(* PLC project SPS_Demonstrator, Beckhoff Automation GmbH TwinCAT PLC Control 3.5.21.30 *)
(* stored: creationDateTime 2026-04-30T11:55:43.4526457, modificationDateTime 2026-04-30T11:55:43.4526457 *)

PROGRAM HRL_SkillSet
VAR
//Hochregallager Skillset	
	//HRL CombinedSkill_Auslagerung
	{attribute 'OPC.UA.DA':= '1'}
	HRL_NMethod_Auslagern : HRL_NMethod_Auslagern;
	bAuslagernAktiv : BOOL := FALSE;
	//HRL Conveyorbelt Skills
	{attribute 'OPC.UA.DA':= '1'}
	HRL_Skill_CB_MoveForwards: HRL_CB_AS_HorizontalMoveSensors; //Movement to Store-Out some goods on the Conveyorbelt
	{attribute 'OPC.UA.DA':= '1'}
	HRL_Skill_CB_MoveBackwards : HRL_CB_AS_HorizontalMoveSensors; //Movement to Store-In some goods on the Conveyorbelt
	
	//HRL RGB Skills
	{attribute 'OPC.UA.DA':= '1'}
	HRL_Skill_RGB_MoveBackwards : HRL_RGB_AS_HorizontalMoveSensors;	
	{attribute 'OPC.UA.DA':= '1'}
	HRL_Skill_RGB_MoveForwards : HRL_RGB_AS_HorizontalMoveSensors;	
	{attribute 'OPC.UA.DA':= '1'}
	HRL_Skill_RGB_MoveVerticalForwards : HRL_RGB_AS_VerticalMoveEncoders;	
	{attribute 'OPC.UA.DA':= '1'}
	HRL_Skill_RGB_MoveVerticalBackwards : HRL_RGB_AS_VerticalMoveEncoders;
	{attribute 'OPC.UA.DA':= '1'}
	HRL_Skill_RGB_MoveHorizontalForwards : HRL_RGB_AS_HorizontalMoveEncoders;	
	{attribute 'OPC.UA.DA':= '1'}
	HRL_Skill_RGB_MoveHorizontalBackwards : HRL_RGB_AS_HorizontalMoveEncoders;
	
	//Organisation FBs
	HRL_ControlOfOutputs : HRL_ControlOfOutputs;
	HRL_OperatingModes : HRL_OperatingModes;
	HRL_DiagnosisHandler : HRL_DiagnosisHandler;
	bAuslagernTrackingLatched : BOOL := FALSE;
	
	//InitialStateDrives
	HRL_RGB_InitialStateDrive : HRL_RGB_InitialStateDrive;
	
	
//Variablen zur Outputsteuerung
	HRL_CB_forwards : BOOL; //GVL_HRL.HRL_MOT_Foerderband_vorwaerts
	HRL_CB_backwards : BOOL; //GVL_HRL.HRL_MOT_Foerderband_rueckwaerts
	HRL_RGB_Forwards01 : BOOL; //GVL_HRL.HRL_MOT_Ausleger_vorwaerts
	HRL_RGB_Forwards02 : BOOL; //GVL_HRL.HRL_MOT_Ausleger_vorwaerts
	HRL_RGB_Backwards01 : BOOL; //GVL_HRL.HRL_MOT_Ausleger_rueckwaerts
	HRL_RGB_Backwards02 : BOOL; //GVL_HRL.HRL_MOT_Ausleger_rueckwaerts	
	HRL_RGB_VertikalDown01 : BOOL; //GVL_HRL.HRL_MOT_vertikal_runter		
	HRL_RGB_VertikalDown02 : BOOL; //GVL_HRL.HRL_MOT_vertikal_runter
	HRL_RGB_VertikalUp01 : BOOL; //GVL_HRL.HRL_MOT_vertikal_hoch
	HRL_RGB_VertikalUp02 : BOOL; //GVL_HRL.HRL_MOT_vertikal_hoch
	HRL_RGB_HorizontalForwards01 : BOOL; //GVL_HRL.HRL_MOT_horizontal_zum_Regal	
	HRL_RGB_HorizontalForwards02 : BOOL; //GVL_HRL.HRL_MOT_horizontal_zum_Regal	
	HRL_RGB_HorizontalBackwards01 : BOOL; //GVL_HRL.HRL_MOT_horizontal_zum_Foerderband
	HRL_RGB_HorizontalBackwards02 : BOOL; //GVL_HRL.HRL_MOT_horizontal_zum_Foerderband
//OutputVariablen für Init-Fahrt	
	Init_SRM_MotorBackwards : BOOL;
	Init_SRM_MotorForwards : BOOL;
	Init_RGB_VerticalUp : BOOL;
	Init_RGB_VerticalDown : BOOL;
	Init_RGB_HorizontalForwards : BOOL;
	Init_RGB_HorizontalBackwards : BOOL;
	
//Time Constraints
	TIME_TSR : TIME := T#150MS;
//Encoder Values for InitialStateDrive
	HRL_RGB_ET_Vertical01 : UDINT;
	HRL_RGB_ET_Vertical02 : UDINT;
	HRL_RGB_ET_Horizontall01 : UDINT;
	HRL_RGB_ET_Horizontall02 : UDINT;
	
	//GEMMA_Mappings
	sCurrentGemmaState : STRING(80) := '';
    sLastNonFailureGemmaState : STRING(80) := '';
    rtD2 : R_TRIG;
END_VAR

VAR_INPUT
	//Variablensetzung: Sollte später über SkillOA eingesetzt werden ODER Hard in SPS codiert (Diskussionspunkt)
	ResetButton: BOOL;
	StartButton: BOOL;
	ConfirmationButton: BOOL;
END_VAR

                  (* === Simulations-Override *)
IF GVL_Sim.bSimMode THEN
    GVL.diNotAus_Kanal_A                  := GVL_Sim.diNotAus_Kanal_A;
    GVL.diNotAus_Kanal_B                  := GVL_Sim.diNotAus_Kanal_B;
    GVL_HRL.HRL_Enc_horizontal_I1          := GVL_HRL_Sim.HRL_Enc_horizontal_I1;
    GVL_HRL.HRL_Enc_horizontal_I2          := GVL_HRL_Sim.HRL_Enc_horizontal_I2;
    GVL_HRL.HRL_Enc_vertikal_I1            := GVL_HRL_Sim.HRL_Enc_vertikal_I1;
    GVL_HRL.HRL_Enc_vertikal_I2            := GVL_HRL_Sim.HRL_Enc_vertikal_I2;
    // GVL_HRL - Digitaleingänge (BOOL)
    GVL_HRL.HRL_Ref_Taster_horizontal      := GVL_HRL_Sim.HRL_Ref_Taster_horizontal;
    GVL_HRL.HRL_LS_innen                   := GVL_HRL_Sim.HRL_LS_innen;
    GVL_HRL.HRL_LS_aussen                  := GVL_HRL_Sim.HRL_LS_aussen;
    GVL_HRL.HRL_Ref_Taster_vertikal        := GVL_HRL_Sim.HRL_Ref_Taster_vertikal;
    GVL_HRL.HRL_Spursensor_1_unten         := GVL_HRL_Sim.HRL_Spursensor_1_unten;
    GVL_HRL.HRL_Spursensor_2_oben          := GVL_HRL_Sim.HRL_Spursensor_2_oben;
    GVL_HRL.HRL_Ref_Taster_Ausleger_vorne  := GVL_HRL_Sim.HRL_Ref_Taster_Ausleger_vorne;
    GVL_HRL.HRL_Ref_Taster_Ausleger_hinten := GVL_HRL_Sim.HRL_Ref_Taster_Ausleger_hinten;
END_IF
(* ============================================================================= *)
HRL_OperatingModes(
    Start := StartButton,
    Stop := NOT (((GVL.diNotAus_Kanal_A) AND (GVL.diNotAus_Kanal_B))),
    Reset := ResetButton,
    Schalter := ConfirmationButton,
    Schrittkette_GS := ((HRL_RGB_InitialStateDrive.ResetMethodCall_SRM) AND (HRL_RGB_InitialStateDrive.ResetMethodCall_RGB_Horizontal) AND (HRL_RGB_InitialStateDrive.ResetMethodCall_RGB_Vertical)),
    Count1 := HRL_RGB_InitialStateDrive.Count_SRM_MotorBackw,
    Count2 := HRL_RGB_InitialStateDrive.Count_SRM_MotorForw,
    Alt_abort := OPCUA.Alt_abort,
    Err_detected := HRL_DiagnosisHandler.Err_detected,
    Diag_finished := HRL_DiagnosisHandler.Diag_finished,
    Alt_found := HRL_DiagnosisHandler.Alt_found,
    Cycle_finished := OPCUA.Cycle_finished
);


HRL_NMethod_Auslagern(
    ESS_OK := ((GVL.diNotAus_Kanal_A) AND (GVL.diNotAus_Kanal_B)),
    AutomaticMode := HRL_OperatingModes.F1,

    HRL_Enc_horizontal_I1 := GVL_HRL.HRL_Enc_horizontal_I1,
    HRL_Enc_horizontal_I2 := GVL_HRL.HRL_Enc_horizontal_I2,
    HRL_Enc_vertikal_I1 := GVL_HRL.HRL_Enc_vertikal_I1,
    HRL_Enc_vertikal_I2 := GVL_HRL.HRL_Enc_vertikal_I2,

    HRL_Ref_Taster_horizontal := GVL_HRL.HRL_Ref_Taster_horizontal,
    HRL_Ref_Taster_vertikal := GVL_HRL.HRL_Ref_Taster_vertikal,
    HRL_Ref_Taster_Ausleger_vorne := GVL_HRL.HRL_Ref_Taster_Ausleger_vorne,
    HRL_Ref_Taster_Ausleger_hinten := GVL_HRL.HRL_Ref_Taster_Ausleger_hinten,

    HRL_LS_innen := GVL_HRL.HRL_LS_innen,
    HRL_LS_aussen := GVL_HRL.HRL_LS_aussen
);

HRL_DiagnosisHandler(
    Diagnose_gefordert := HRL_OperatingModes.D2,
    ErrorDetectedRaw := HRL_NMethod_Auslagern.Error,
    Reset := ResetButton
);

HRL_RGB_InitialStateDrive(
    MethodCall_InitDrive := HRL_OperatingModes.MethodCall_InitStateDrive,
    ESS := ((GVL.diNotAus_Kanal_A) AND (GVL.diNotAus_Kanal_B)),
    InputInitDriveMode := HRL_OperatingModes.InputVar_InitStateDrive,
    TouchSensor01_SRM := GVL_HRL.HRL_Ref_Taster_Ausleger_hinten,
    TouchSensor02_RGB_vertical := GVL_HRL.HRL_Ref_Taster_vertikal,
    TouchSensor03_RGB_horizontal := GVL_HRL.HRL_Ref_Taster_horizontal,
    TOF_Time_TSR := TIME_TSR,
    InitDriveMode := HRL_OperatingModes.A6
);
Init_SRM_MotorBackwards := HRL_RGB_InitialStateDrive.SRM_MotorBackwards;
HRL_Skill_CB_MoveForwards(
    ESS := ((GVL.diNotAus_Kanal_A) AND (GVL.diNotAus_Kanal_B)),
    LightBarrierSensor_01 := GVL_HRL.HRL_LS_innen,
    LightBarrierSensor_02 := GVL_HRL.HRL_LS_aussen,
    AutomaticMode := HRL_OperatingModes.F1
);
HRL_CB_forwards := HRL_Skill_CB_MoveForwards.DO_MovingConveyorBelt;
HRL_Skill_CB_MoveBackwards(
    ESS := ((GVL.diNotAus_Kanal_A) AND (GVL.diNotAus_Kanal_B)),
    LightBarrierSensor_01 := GVL_HRL.HRL_LS_aussen,
    LightBarrierSensor_02 := GVL_HRL.HRL_LS_innen,
    AutomaticMode := HRL_OperatingModes.F1
);
HRL_CB_backwards := HRL_Skill_CB_MoveBackwards.DO_MovingConveyorBelt;
HRL_Skill_RGB_MoveForwards(
    ESS := ((GVL.diNotAus_Kanal_A) AND (GVL.diNotAus_Kanal_B)),
    TouchSensor01 := GVL_HRL.HRL_Ref_Taster_Ausleger_hinten,
    TouchSensor02 := GVL_HRL.HRL_Ref_Taster_Ausleger_vorne,
    TOF_Time_TSR := TIME_TSR,
    AutomaticMode := HRL_OperatingModes.F1
);
HRL_RGB_Forwards01 := HRL_Skill_RGB_MoveForwards.DO_MovingHorizontalRGB_01;
HRL_Skill_RGB_MoveBackwards(
    ESS := ((GVL.diNotAus_Kanal_A) AND (GVL.diNotAus_Kanal_B)),
    TouchSensor01 := GVL_HRL.HRL_Ref_Taster_Ausleger_vorne,
    TouchSensor02 := GVL_HRL.HRL_Ref_Taster_Ausleger_hinten,
    TOF_Time_TSR := TIME_TSR,
    AutomaticMode := HRL_OperatingModes.F1
);
HRL_RGB_Backwards01 := HRL_Skill_RGB_MoveBackwards.DO_MovingHorizontalRGB_01;
HRL_Skill_RGB_MoveVerticalForwards(
    ESS := ((GVL.diNotAus_Kanal_A) AND (GVL.diNotAus_Kanal_B)),
    TouchSensor01 := GVL_HRL.HRL_Ref_Taster_vertikal,
    EncoderStartPosition01 := GVL_HRL.HRL_Enc_vertikal_I1,
    EncoderStartPosition02 := GVL_HRL.HRL_Enc_vertikal_I2,
    TOF_TSR_TIME := TIME_TSR,
    AutomaticMode := HRL_OperatingModes.F1
);
HRL_RGB_VertikalDown01 := HRL_Skill_RGB_MoveVerticalForwards.DO_MovingVerticalRGB_01;
HRL_Skill_RGB_MoveVerticalBackwards(
    ESS := ((GVL.diNotAus_Kanal_A) AND (GVL.diNotAus_Kanal_B)),
    TouchSensor01 := GVL_HRL.HRL_Ref_Taster_vertikal,
    EncoderStartPosition01 := GVL_HRL.HRL_Enc_vertikal_I1,
    EncoderStartPosition02 := GVL_HRL.HRL_Enc_vertikal_I2,
    TOF_TSR_TIME := TIME_TSR,
    AutomaticMode := HRL_OperatingModes.F1
);
HRL_RGB_VertikalUp02 := HRL_Skill_RGB_MoveVerticalBackwards.DO_MovingVerticalRGB_01;
HRL_Skill_RGB_MoveHorizontalForwards(
    ESS := ((GVL.diNotAus_Kanal_A) AND (GVL.diNotAus_Kanal_B)),
    TouchSensor01 := GVL_HRL.HRL_Ref_Taster_horizontal,
    EncoderStartPosition01 := GVL_HRL.HRL_Enc_horizontal_I1,
    EncoderStartPosition02 := GVL_HRL.HRL_Enc_horizontal_I2,
    TOF_Time_TSR := TIME_TSR,
    AutomaticMode := HRL_OperatingModes.F1
);
HRL_RGB_HorizontalForwards01 := HRL_Skill_RGB_MoveHorizontalForwards.DO_MovingHorizontalRGB_01;
HRL_Skill_RGB_MoveHorizontalBackwards(
    ESS := ((GVL.diNotAus_Kanal_A) AND (GVL.diNotAus_Kanal_B)),
    TouchSensor01 := GVL_HRL.HRL_Ref_Taster_horizontal,
    EncoderStartPosition01 := GVL_HRL.HRL_Enc_horizontal_I1,
    EncoderStartPosition02 := GVL_HRL.HRL_Enc_horizontal_I2,
    TOF_Time_TSR := TIME_TSR,
    AutomaticMode := HRL_OperatingModes.F1
);
HRL_RGB_HorizontalBackwards02 := HRL_Skill_RGB_MoveHorizontalBackwards.DO_MovingHorizontalRGB_01;

bAuslagernAktiv := HRL_NMethod_Auslagern.Busy OR (HRL_NMethod_Auslagern.CurrentStep <> 0);;

HRL_ControlOfOutputs(
    F4 := HRL_OperatingModes.F4,
    F1 := HRL_OperatingModes.F1,
    A2 := HRL_OperatingModes.A2,
    A1 := HRL_OperatingModes.A1,
    A6 := HRL_OperatingModes.A6,
    Start := HRL_OperatingModes.Start,

    CB_forwards :=
        (HRL_CB_forwards AND NOT bAuslagernAktiv)
        OR HRL_NMethod_Auslagern.REQ_CB_forwards,

    CB_backwards :=
        (HRL_CB_backwards AND NOT bAuslagernAktiv)
        OR HRL_NMethod_Auslagern.REQ_CB_backwards,

    RGB_Forwards01 :=
        (HRL_RGB_Forwards01 AND NOT bAuslagernAktiv)
        OR HRL_NMethod_Auslagern.REQ_RGB_Forwards,

    RGB_Forwards02 :=
        HRL_RGB_Forwards02 AND NOT bAuslagernAktiv,

    RGB_Backwards01 :=
        (HRL_RGB_Backwards01 AND NOT bAuslagernAktiv)
        OR HRL_NMethod_Auslagern.REQ_RGB_Backwards,

    RGB_Backwards02 :=
        HRL_RGB_Backwards02 AND NOT bAuslagernAktiv,

    RGB_VertikalDown01 :=
        (HRL_RGB_VertikalDown01 AND NOT bAuslagernAktiv)
        OR HRL_NMethod_Auslagern.REQ_RGB_VerticalDown,

    RGB_VertikalDown02 :=
        HRL_RGB_VertikalDown02 AND NOT bAuslagernAktiv,

    RGB_VertikalUp01 :=
        (HRL_RGB_VertikalUp01 AND NOT bAuslagernAktiv)
        OR HRL_NMethod_Auslagern.REQ_RGB_VerticalUp,

    RGB_VertikalUp02 :=
        HRL_RGB_VertikalUp02 AND NOT bAuslagernAktiv,

    RGB_HorizontalForwards01 :=
        (HRL_RGB_HorizontalForwards01 AND NOT bAuslagernAktiv)
        OR HRL_NMethod_Auslagern.REQ_RGB_HorizontalForward,

    RGB_HorizontalForwards02 :=
        HRL_RGB_HorizontalForwards02 AND NOT bAuslagernAktiv,

    RGB_HorizontalBackwards01 :=
        (HRL_RGB_HorizontalBackwards01 AND NOT bAuslagernAktiv)
        OR HRL_NMethod_Auslagern.REQ_RGB_HorizontalBackward,

    RGB_HorizontalBackwards02 :=
        HRL_RGB_HorizontalBackwards02 AND NOT bAuslagernAktiv,

    Init_RGB_Forwards := Init_SRM_MotorForwards,
    Init_RGB_Backwards := Init_SRM_MotorBackwards,
    Init_RGB_VertikalUp := Init_RGB_VerticalUp,
    Init_RGB_VertikalDown := Init_RGB_VerticalDown,
    Init_RGB_HorizontalForwads := Init_RGB_HorizontalForwards,
    Init_RGB_HorizontalBackwards := Init_RGB_HorizontalBackwards
);
IF GVL_Sim.bSimMode THEN

    // Outputs in Simulationsabbild schreiben
    GVL_HRL_Sim.HRL_MOT_Foerderband_vorwaerts :=
        HRL_ControlOfOutputs.ConveyorBeltForward;

    GVL_HRL_Sim.HRL_MOT_Foerderband_rueckwaerts :=
        HRL_ControlOfOutputs.ConveyorBeltBackward;

    GVL_HRL_Sim.HRL_MOT_Ausleger_vorwaerts :=
        HRL_ControlOfOutputs.RGB_Forwards;

    GVL_HRL_Sim.HRL_MOT_Ausleger_rueckwaerts :=
        HRL_ControlOfOutputs.RGB_Backwards;

    GVL_HRL_Sim.HRL_MOT_vertikal_runter :=
        HRL_ControlOfOutputs.RGB_VerticalDown;

    GVL_HRL_Sim.HRL_MOT_vertikal_hoch :=
        HRL_ControlOfOutputs.RGB_VerticalUp;

    GVL_HRL_Sim.HRL_MOT_horizontal_zum_Regal :=
        HRL_ControlOfOutputs.RGB_HorizontalForward;

    GVL_HRL_Sim.HRL_MOT_horizontal_zum_Foerderband :=
        HRL_ControlOfOutputs.RGB_HorizontalBackward;

    GVL_HRL_Sim.HRL_K1_1_Zaehler_Zuruecksetzen :=
        GVL_HRL.HRL_K1_1_Zaehler_Zuruecksetzen;

    GVL_HRL_Sim.HRL_K1_2_Zaehler_Zuruecksetzen :=
        GVL_HRL.HRL_K1_2_Zaehler_Zuruecksetzen;

ELSE

    // Outputs auf reale Hardware schreiben
    GVL_HRL.HRL_MOT_Foerderband_vorwaerts :=
        HRL_ControlOfOutputs.ConveyorBeltForward;

    GVL_HRL.HRL_MOT_Foerderband_rueckwaerts :=
        HRL_ControlOfOutputs.ConveyorBeltBackward;

    GVL_HRL.HRL_MOT_Ausleger_vorwaerts :=
        HRL_ControlOfOutputs.RGB_Forwards;

    GVL_HRL.HRL_MOT_Ausleger_rueckwaerts :=
        HRL_ControlOfOutputs.RGB_Backwards;

    GVL_HRL.HRL_MOT_vertikal_runter :=
        HRL_ControlOfOutputs.RGB_VerticalDown;

    GVL_HRL.HRL_MOT_vertikal_hoch :=
        HRL_ControlOfOutputs.RGB_VerticalUp;

    GVL_HRL.HRL_MOT_horizontal_zum_Regal :=
        HRL_ControlOfOutputs.RGB_HorizontalForward;

    GVL_HRL.HRL_MOT_horizontal_zum_Foerderband :=
        HRL_ControlOfOutputs.RGB_HorizontalBackward;

END_IF;

//GEMMA-Mappings
IF HRL_OperatingModes.A1 THEN
    sCurrentGemmaState := 'HRL_OperatingModes.A1';
ELSIF HRL_OperatingModes.A2 THEN
    sCurrentGemmaState := 'HRL_OperatingModes.A2';
ELSIF HRL_OperatingModes.A5 THEN
    sCurrentGemmaState := 'HRL_OperatingModes.A5';
ELSIF HRL_OperatingModes.A6 THEN
    sCurrentGemmaState := 'HRL_OperatingModes.A6';
ELSIF HRL_OperatingModes.F1 THEN
    sCurrentGemmaState := 'HRL_OperatingModes.F1';
ELSIF HRL_OperatingModes.F4 THEN
    sCurrentGemmaState := 'HRL_OperatingModes.F4';
ELSIF HRL_OperatingModes.D1 THEN
    sCurrentGemmaState := 'HRL_OperatingModes.D1';
ELSIF HRL_OperatingModes.D3 THEN
    sCurrentGemmaState := 'HRL_OperatingModes.D3';
END_IF;

IF NOT HRL_OperatingModes.D2 THEN
    sLastNonFailureGemmaState := sCurrentGemmaState;
END_IF;

rtD2(CLK := HRL_OperatingModes.D2);

IF rtD2.Q THEN
    OPCUA.LastGEMMAStateBeforeFailure := sLastNonFailureGemmaState;
END_IF;
                
END_PROGRAM

PROGRAM MBS_SkillSet
VAR
//Multibearbeitungsstation Skills
	//MBS Maschine1 (Ofen) Skills	
	{attribute 'OPC.UA.DA':= '1'}
	MBS_Skill_MR01_TransportIn: MBS_MR01_AS_HorizontalMoveSensors;
	{attribute 'OPC.UA.DA':= '1'}
	MBS_Skill_MR01_SecuringWorkpiece: MBS_MR01_AS_SecuringProcess;
	{attribute 'OPC.UA.DA':= '1'}
	MBS_Skill_MR01_HardeningProcess: MBS_MR01_AS_HardeningProcess;
	{attribute 'OPC.UA.DA':= '1'}
	MBS_SkillMR01_ReleaseWorkpiece: MBS_MR01_AS_SecuringProcess;
	{attribute 'OPC.UA.DA':= '1'}
	MBS_Skill_MR01_TransportOut: MBS_MR01_AS_HorizontalMoveSensors;
	
	//MBS Vakuumsauggreifer Skills
	{attribute 'OPC.UA.DA':= '1'}
	MBS_Skill_VGS_PickUpWorkpieceToDmPD: MBS_VSG_AS_SuctionProcess;
	{attribute 'OPC.UA.DA':= '1'}
	MBS_Skill_VGS_PickUpWorkpieceToOven: MBS_VSG_AS_SuctionProcess;
	{attribute 'OPC.UA.DA':= '1'}
	MBS_Skill_VSG_VerticalMove: MBS_VSG_AS_VerticalMove;	
	{attribute 'OPC.UA.DA':= '1'}
	MBS_Skill_VSG_TransportToDmPD: MBS_VSG_AS_HorizontalMove;
	{attribute 'OPC.UA.DA':= '1'}
	MBS_Skill_VSG_TransportToMR01: MBS_VSG_AS_HorizontalMove;
	
	
	//MBS Drehteller mit PushingDevice Skills
	{attribute 'OPC.UA.DA':= '1'}
	MBS_Skill_DmPD_RotateFromVSGtoMR02: MBS_DmPD_AS_RotationMove;
	{attribute 'OPC.UA.DA':= '1'}
	MBS_Skill_DmPD_RotateFromVSGtoCB: MBS_DmPD_AS_RotationMove;
	{attribute 'OPC.UA.DA':= '1'}
	MBS_Skill_DmPD_RotateFromMR02toCB: MBS_DmPD_AS_RotationMove;
	{attribute 'OPC.UA.DA':= '1'}
	MBS_Skill_DmPD_RotateFromMR02toVSG: MBS_DmPD_AS_RotationMove;
	{attribute 'OPC.UA.DA':= '1'}
	MBS_Skill_DmPD_RotateFromCBtoVSG: MBS_DmPD_AS_RotationMove;
	{attribute 'OPC.UA.DA':= '1'}
	MBS_Skill_DmPD_RotateFromCBtoMR02: MBS_DmPD_AS_RotationMove;
	{attribute 'OPC.UA.DA':= '1'}
	MBS_Skill_DmPB_PushWorkpieceOff: MBS_DmPD_AS_HorizontalMove;
	
	//MBS Maschine2 (Schneidemaschine) Skills
	{attribute 'OPC.UA.DA':= '1'}
	MBS_Skill_MR02_CuttingProcess: MBS_MR02_AS_CuttingProcess;
	
	//MBS ConveyorBelt Skills
	{attribute 'OPC.UA.DA':= '1'}
	MBS_Skill_CB_Moving: MBS_CB_AS_HorizontalMove;
	
	//Organisation FBs
	MBS_ControlOfOutputs : MBS_ControlOfOutputs;
	MBS_OperatingModes : MBS_OperatingModes;
	
	//InitialStateDrives
	MBS_MR01_InitialStateDrive : MBS_MR01_InitialStateDrive;
	MBS_VSG_InitialStateDrive : MBS_VSG_InitialStateDrive;
	MBS_DmPD_InitialStateDrive : MBS_DmPD_InitialStateDrive;
	MBS_MR02_InitialStateDrive : MBS_MR02_InitialStateDrive;
	
//Variablen zur Outputsteuerung
	//Output-Variablen der Komponente MR01 
	MR01_MoveOvenslideIn 			: BOOL; //GVL_MBS.MBS_MOT_Ofenschieber_einfahren
	MR01_MoveOvenslideOut			: BOOL; //GVL_MBS.MBS_MOT_Ofenschieber_ausfahren
	MR01_Compressor_SecuringProcess : BOOL; //GVL_MBS.MBS_Kompressor
	MR01_Valve_OvenDoor				: BOOL; //GVL_MBS.MBS_MV_Ofentuer
	MR01_HardeningProcess			: BOOL; //GVL_MBS.MBS_Leuchte_Ofen
	
	//Output-Variablen der Komponente VSG
	VSG_Compressor_VerticalMove			: BOOL; //GVL_MBS.MBS_Kompressor
	VSG_Valve_VerticalMove				: BOOL; //GVL_MBS.MBS_MV_senken
	VSG_Compressor_SuctionProcessToDmPD	: BOOL; //GVL_MBS.MBS_Kompressor
	VSG_Valve_SuctionProcessToDmPD		: BOOL; //GVL_MBS.MBS_MV_Vakuum
	VSG_Compressor_SuctionProcessToMR01	: BOOL; //GVL_MBS.MBS_Kompressor
	VSG_Valve_SuctionProcessToMR01		: BOOL; //GVL_MBS.MBS_MV_Vakuum
	VSG_MoveHorizontalForwards			: BOOL; //GVL_MBS.MBS_MOT_Sauger_zum_DK
	VSG_MoveHorizontalBackwards			: BOOL; //GVL_MBS.MBS_MOT_Sauger_zum_Ofen
		
	//Output-Variablen der Komponente DmPD
	DmPD_RotateCWformVSGtoMR02 		: BOOL; //GVL_MBS.MBS_MOT_DK_CW
	DmPD_RotateCWromVSGtoCB			: BOOL; //GVL_MBS.MBS_MOT_DK_CW
	DmPD_RotateCWfromMR02toCB		: BOOL; //GVL_MBS.MBS_MOT_DK_CW
	DmPD_RotateCCWformCBtoMR02 		: BOOL; //GVL_MBS.MBS_MOT_DK_CCW
	DmPD_RotateCCWformCBtoVSG 		: BOOL; //GVL_MBS.MBS_MOT_DK_CCW
	DmPD_RotateCCWformMR02toVSG 	: BOOL; //GVL_MBS.MBS_MOT_DK_CCW
	DmPD_Compressor_HorizontalMove 	: BOOL; //GVL_MBS.MBS_Kompressor
	DmPD_Valve_HorizontalMove 		: BOOL; //GVL_MBS.ControlValveHorizontalMove
	
	//Output-Variablen der Komponente MR02
	MR02_CuttingProcess : BOOL; //GVL_MBS.MBS_MOT_Saege
	
	//Output-Variablen der Komponente CB
	CB_MoveForwards	: BOOL; //GVL_MBS.MBS_MOT_Foerderband_vorwaerts
	
//Output-Variablen für Init-Fahrt
	Init_MR01_HorizontalForwards	: BOOL; //GVL_MBS.MBS_MOT_Ofenschieber_einfahren
	Init_MR01_HorizontalBackwards	: BOOL; //GVL_MBS.MBS_MOT_Ofenschieber_ausfahren
	Init_VSG_HorizontalForwards 	: BOOL; //GVL_MBS.MBS_MOT_Sauger_zum_DK
	Init_VSG_HorizontalBackwards	: BOOL; //GVL_MBS.MBS_MOT_Sauger_zum_Ofen
	Init_DmPD_RotateCW				: BOOL; //GVL_MBS.MBS_MOT_DK_CW
	Init_DmPD_RotateCCW				: BOOL; //GVL_MBS.MBS_MOT_DK_CCW
	Init_MR02_CuttingProcess		: BOOL; //GVL_MBS.MBS_MOT_Saege
	
//Variablensetzung: Sollte später über SkillOA eingesetzt werden ODER Hard in SPS codiert (Diskussionspunkt)
	ResetButton: BOOL;
	StartButton: BOOL;
	ConfirmationButton: BOOL;

//Time Constraints
	TIME_TSR : TIME := T#150MS;
	PowerOnDelay_Compressor : TIME := T#500MS;
	PowerOnDelay_Valve_SuctionProcess : TIME := T#520MS;
	PowerOnDelay_Valve_VerticalMove : TIME := T#120MS;
	PowerOnDelay_Valve_HorizontalMove : TIME := T#120MS;
	PowerOffDelay_ConveyorBelt : TIME := T#100MS;	
//Encoder Values for InitialStateDrive
	
//Variable Values for InitialStateDrive
	MethodCall_InitStateDrive	: BOOL;
	InputVar_InitStateDrive		: BOOL;
	InitTime_Cutting 			: TIME := T#200MS;

END_VAR

                  MBS_OperatingModes(
    Start := StartButton,
    Stop := ((GVL.diNotAus_Kanal_A) AND (GVL.diNotAus_Kanal_B)),
    Reset := ResetButton,
    Schalter := ConfirmationButton,
    Schrittkette_GS := (((MBS_MR01_InitialStateDrive.ResetMethodCallInitDriveMR01_Backwards) AND (MBS_MR01_InitialStateDrive.ResetMethodCallInitDriveMR01_Forwards) AND (MBS_VSG_InitialStateDrive.ResetMethodCallInitDriveVSG) AND (MBS_DmPD_InitialStateDrive.ResetMethodCallRotateCCW) AND (MBS_DmPD_InitialStateDrive.ResetMethodCallRotateCW) AND (MBS_MR02_InitialStateDrive.ResetMethodCallCuttingProcess)))
);
MBS_ControlOfOutputs(
    F4 := MBS_OperatingModes.F4,
    F1 := MBS_OperatingModes.F1,
    A2 := MBS_OperatingModes.A2,
    A1 := MBS_OperatingModes.A1,
    A6 := MBS_OperatingModes.A6,
    Start := MBS_OperatingModes.Start,
    CB_Forwards := CB_MoveForwards,
    DmPD_Compressor := DmPD_Compressor_HorizontalMove,
    DmPD_Valve := DmPD_Valve_HorizontalMove,
    DmPD_RotateCW_VSGtoMR02 := DmPD_RotateCWformVSGtoMR02,
    DmPD_RotateCW_VSGtoCB := DmPD_RotateCWromVSGtoCB,
    DmPD_RotateCW_MR02toCB := DmPD_RotateCWfromMR02toCB,
    DmPD_RotateCCW_CBtoMR02 := DmPD_RotateCCWformCBtoMR02,
    DmPD_RotateCCW_CBtoVSG := DmPD_RotateCCWformCBtoVSG,
    DmPD_RotateCCW_MR02toVSG := DmPD_RotateCCWformMR02toVSG,
    MR01_HardeningProcess := MR01_HardeningProcess,
    MR01_HorizontalForwards := MR01_MoveOvenslideIn,
    MR01_HoritzontalBackwards := MR01_MoveOvenslideOut,
    MR01_Compressor := MR01_Compressor_SecuringProcess,
    MR01_Valve := MR01_Valve_OvenDoor,
    MR02_CuttingProcess := MR02_CuttingProcess,
    VSG_HorizontalForwards := VSG_MoveHorizontalForwards,
    VSG_HorizontalBackwards := VSG_MoveHorizontalBackwards,
    VSG_Valve_VerticalDown := VSG_Valve_VerticalMove,
    VSG_Valve_SuctionToDmPD := VSG_Valve_SuctionProcessToDmPD,
    VSG_Valve_SuctionToMR01 := VSG_Valve_SuctionProcessToMR01,
    VSG_Compressor_VerticalDown := VSG_Compressor_VerticalMove,
    VSG_Compressor_SuctionToDmPD := VSG_Compressor_SuctionProcessToDmPD,
    VSG_Compressor_SuctionToMR01 := VSG_Compressor_SuctionProcessToMR01,
    Init_DmPD_RotateCCW := Init_DmPD_RotateCCW,
    Init_DmPD_RotateCW := Init_DmPD_RotateCW,
    Init_MR01_HorizontalForwards := Init_MR01_HorizontalForwards,
    Init_MR01_HorizontalBackwards := Init_MR01_HorizontalBackwards,
    Init_MR02_CuttingProcess := Init_MR02_CuttingProcess,
    Init_VSG_HorizontalForwards := Init_VSG_HorizontalForwards,
    Init_VSG_HorizontalBackwards := Init_VSG_HorizontalBackwards
);
GVL_MBS.MBS_MOT_Foerderband_vorwaerts := MBS_ControlOfOutputs.ConveyorBeltForward;
MBS_MR01_InitialStateDrive(
    MethodCall_InitDrive := MethodCall_InitStateDrive,
    ESS := ((GVL.diNotAus_Kanal_A) AND (GVL.diNotAus_Kanal_B)),
    InputInitStateDrive := InputVar_InitStateDrive,
    TouchSensor01 := GVL_MBS.MBS_Ref_Taster_Ofenschieber_innen,
    TouchSensor02 := GVL_MBS.MBS_Ref_Taster_Ofenschieber_aussen,
    InitDriveMode := MBS_OperatingModes.A6
);
Init_MR01_HorizontalForwards := MBS_MR01_InitialStateDrive.MotorControlHorizontalForwards;
MBS_VSG_InitialStateDrive(
    MethodCall_InitDrive := MethodCall_InitStateDrive,
    ESS := ((GVL.diNotAus_Kanal_A) AND (GVL.diNotAus_Kanal_B)),
    InputInitStateDrive := InputVar_InitStateDrive,
    TouchSensor01 := GVL_MBS.MBS_Ref_Taster_Sauger_Pos_DK,
    TOF_Time_TSR := TIME_TSR,
    InitDriveMode := MBS_OperatingModes.A6
);
Init_VSG_HorizontalForwards := MBS_VSG_InitialStateDrive.DO_HorizontalMoveInitDriveVSG_01;
MBS_DmPD_InitialStateDrive(
    MethodCall_InitDrive := MethodCall_InitStateDrive,
    ESS := ((GVL.diNotAus_Kanal_A) AND (GVL.diNotAus_Kanal_B)),
    InputInitialStateDrive := InputVar_InitStateDrive,
    DI02_CW := GVL_MBS.MBS_Ref_Taster_DK_Pos_Foerderband,
    DI01_CCW := GVL_MBS.MBS_Ref_Taster_DK_Pos_Foerderband,
    DI02_CCW := GVL_MBS.MBS_Ref_Taster_DK_Pos_Sauger,
    InitDriveMode := MBS_OperatingModes.A6
);
Init_DmPD_RotateCW := MBS_DmPD_InitialStateDrive.MotorControl_CW;
MBS_MR02_InitialStateDrive(
    MethodCall_InitDrive := MethodCall_InitStateDrive,
    ESS := ((GVL.diNotAus_Kanal_A) AND (GVL.diNotAus_Kanal_B)),
    InputInitialStateDrive := InputVar_InitStateDrive,
    TOF_Time_InitCuttingTime := InitTime_Cutting,
    InitDriveMode := MBS_OperatingModes.A6
);
Init_MR02_CuttingProcess := MBS_MR02_InitialStateDrive.CheckMR02MotorControl;
MBS_Skill_MR01_TransportIn(
    ESS := ((GVL.diNotAus_Kanal_A) AND (GVL.diNotAus_Kanal_B)),
    TouchSensor_01 := GVL_MBS.MBS_Ref_Taster_Ofenschieber_aussen,
    TouchSensor_02 := GVL_MBS.MBS_Ref_Taster_Ofenschieber_innen,
    TOF_Time_TSR := TIME_TSR,
    AutomaticMode := MBS_OperatingModes.F1
);
MR01_MoveOvenslideIn := MBS_Skill_MR01_TransportIn.DO_MovingHorizontalMR01_01;
MBS_Skill_MR01_TransportOut(
    ESS := ((GVL.diNotAus_Kanal_A) AND (GVL.diNotAus_Kanal_B)),
    TouchSensor_01 := GVL_MBS.MBS_Ref_Taster_Ofenschieber_innen,
    TouchSensor_02 := GVL_MBS.MBS_Ref_Taster_Ofenschieber_aussen,
    TOF_Time_TSR := TIME_TSR,
    AutomaticMode := MBS_OperatingModes.F1
);
MR01_MoveOvenslideOut := MBS_Skill_MR01_TransportOut.DO_MovingHorizontalMR01_01;
MBS_Skill_MR01_SecuringWorkpiece(ESS := ((GVL.diNotAus_Kanal_A) AND (GVL.diNotAus_Kanal_B)), TouchSensor_01 := GVL_MBS.MBS_Ref_Taster_Ofenschieber_innen, AutomaticMode := MBS_OperatingModes.F1);
MR01_Compressor_SecuringProcess := MBS_Skill_MR01_SecuringWorkpiece.DO_SecuringProcessCompressorMR01_01;
MBS_Skill_MR01_HardeningProcess(ESS := ((GVL.diNotAus_Kanal_A) AND (GVL.diNotAus_Kanal_B)), LightSensor_01 := GVL_MBS.MBS_Ref_Taster_Ofenschieber_innen, AutomaticMode := MBS_OperatingModes.F1);
MR01_HardeningProcess := MBS_Skill_MR01_HardeningProcess.DO_HardeningProcessControlMR01;
MBS_Skill_VSG_VerticalMove(
    ESS := ((GVL.diNotAus_Kanal_A) AND (GVL.diNotAus_Kanal_B)),
    TouchSensor_01 := GVL_MBS.MBS_Ref_Taster_Sauger_Pos_DK,
    TON_PowerOnDelay_Compressor := PowerOnDelay_Compressor,
    TON_PowerOnDelay_Valve := PowerOnDelay_Valve_VerticalMove,
    AutomaticMode := MBS_OperatingModes.F1
);
VSG_Compressor_VerticalMove := MBS_Skill_VSG_VerticalMove.DO_ControlCompressorVerticalMoveVSG_01;
MBS_Skill_VGS_PickUpWorkpieceToDmPD(
    ESS := ((GVL.diNotAus_Kanal_A) AND (GVL.diNotAus_Kanal_B)),
    TouchSensor_01 := GVL_MBS.MBS_Ref_Taster_Sauger_Pos_Ofen,
    TouchSensor_02 := GVL_MBS.MBS_Ref_Taster_Sauger_Pos_DK,
    TON_PowerOnDelay_Compressor := PowerOnDelay_Compressor,
    TON_PowerOnDelay_Valve := PowerOnDelay_Valve_SuctionProcess,
    AutomaticMode := MBS_OperatingModes.F1
);
VSG_Compressor_SuctionProcessToDmPD := MBS_Skill_VGS_PickUpWorkpieceToDmPD.DO_ControlCompressorSuctionProcessVSG_01;
MBS_Skill_VGS_PickUpWorkpieceToOven(
    ESS := ((GVL.diNotAus_Kanal_A) AND (GVL.diNotAus_Kanal_B)),
    TouchSensor_01 := GVL_MBS.MBS_Ref_Taster_Sauger_Pos_DK,
    TouchSensor_02 := GVL_MBS.MBS_Ref_Taster_Sauger_Pos_Ofen,
    TON_PowerOnDelay_Compressor := PowerOnDelay_Compressor,
    TON_PowerOnDelay_Valve := PowerOnDelay_Valve_SuctionProcess,
    AutomaticMode := MBS_OperatingModes.F1
);
VSG_Compressor_SuctionProcessToMR01 := MBS_Skill_VGS_PickUpWorkpieceToOven.DO_ControlCompressorSuctionProcessVSG_01;
MBS_Skill_VSG_TransportToDmPD(
    ESS := ((GVL.diNotAus_Kanal_A) AND (GVL.diNotAus_Kanal_B)),
    TouchSensor_01 := GVL_MBS.MBS_Ref_Taster_Sauger_Pos_Ofen,
    TouchSensor_02 := GVL_MBS.MBS_Ref_Taster_Sauger_Pos_DK,
    TOF_Time_TSR := TIME_TSR,
    AutomaticeMode := MBS_OperatingModes.F1
);
VSG_MoveHorizontalForwards := MBS_Skill_VSG_TransportToDmPD.DO_HorizontalMoveVSG_01;
MBS_Skill_VSG_TransportToMR01(
    ESS := ((GVL.diNotAus_Kanal_A) AND (GVL.diNotAus_Kanal_B)),
    TouchSensor_01 := GVL_MBS.MBS_Ref_Taster_Sauger_Pos_DK,
    TouchSensor_02 := GVL_MBS.MBS_Ref_Taster_Sauger_Pos_Ofen,
    TOF_Time_TSR := TIME_TSR,
    AutomaticeMode := MBS_OperatingModes.F1
);
VSG_MoveHorizontalBackwards := MBS_Skill_VSG_TransportToMR01.DO_HorizontalMoveVSG_01;
MBS_Skill_DmPD_RotateFromVSGtoMR02(
    ESS := ((GVL.diNotAus_Kanal_A) AND (GVL.diNotAus_Kanal_B)),
    TouchSensor_01 := GVL_MBS.MBS_Ref_Taster_DK_Pos_Sauger,
    TouchSensor_02 := GVL_MBS.MBS_Ref_Taster_DK_Pos_Saege,
    AutomaticMode := MBS_OperatingModes.F1
);
DmPD_RotateCWformVSGtoMR02 := MBS_Skill_DmPD_RotateFromVSGtoMR02.DO_MovingRotationPmPD_01;
MBS_Skill_DmPD_RotateFromVSGtoCB(
    ESS := ((GVL.diNotAus_Kanal_A) AND (GVL.diNotAus_Kanal_B)),
    TouchSensor_01 := GVL_MBS.MBS_Ref_Taster_DK_Pos_Sauger,
    TouchSensor_02 := GVL_MBS.MBS_Ref_Taster_DK_Pos_Foerderband,
    AutomaticMode := MBS_OperatingModes.F1
);
DmPD_RotateCWromVSGtoCB := MBS_Skill_DmPD_RotateFromVSGtoCB.DO_MovingRotationPmPD_01;
MBS_Skill_DmPD_RotateFromMR02toCB(
    ESS := ((GVL.diNotAus_Kanal_A) AND (GVL.diNotAus_Kanal_B)),
    TouchSensor_01 := GVL_MBS.MBS_Ref_Taster_DK_Pos_Saege,
    TouchSensor_02 := GVL_MBS.MBS_Ref_Taster_DK_Pos_Foerderband,
    AutomaticMode := MBS_OperatingModes.F1
);
DmPD_RotateCWfromMR02toCB := MBS_Skill_DmPD_RotateFromMR02toCB.DO_MovingRotationPmPD_01;
MBS_Skill_DmPD_RotateFromCBtoMR02(
    ESS := ((GVL.diNotAus_Kanal_A) AND (GVL.diNotAus_Kanal_B)),
    TouchSensor_01 := GVL_MBS.MBS_Ref_Taster_DK_Pos_Foerderband,
    TouchSensor_02 := GVL_MBS.MBS_Ref_Taster_DK_Pos_Saege,
    AutomaticMode := MBS_OperatingModes.F1
);
DmPD_RotateCCWformCBtoMR02 := MBS_Skill_DmPD_RotateFromCBtoMR02.DO_MovingRotationPmPD_01;
MBS_Skill_DmPD_RotateFromCBtoVSG(
    ESS := ((GVL.diNotAus_Kanal_A) AND (GVL.diNotAus_Kanal_B)),
    TouchSensor_01 := GVL_MBS.MBS_Ref_Taster_DK_Pos_Foerderband,
    TouchSensor_02 := GVL_MBS.MBS_Ref_Taster_DK_Pos_Sauger,
    AutomaticMode := MBS_OperatingModes.F1
);
DmPD_RotateCCWformCBtoVSG := MBS_Skill_DmPD_RotateFromCBtoVSG.DO_MovingRotationPmPD_01;
MBS_Skill_DmPD_RotateFromMR02toVSG(
    ESS := ((GVL.diNotAus_Kanal_A) AND (GVL.diNotAus_Kanal_B)),
    TouchSensor_01 := GVL_MBS.MBS_Ref_Taster_DK_Pos_Saege,
    TouchSensor_02 := GVL_MBS.MBS_Ref_Taster_DK_Pos_Sauger,
    AutomaticMode := MBS_OperatingModes.F1
);
DmPD_RotateCCWformMR02toVSG := MBS_Skill_DmPD_RotateFromMR02toVSG.DO_MovingRotationPmPD_01;
MBS_Skill_DmPB_PushWorkpieceOff(
    ESS := ((GVL.diNotAus_Kanal_A) AND (GVL.diNotAus_Kanal_B)),
    TouchSensor_01 := GVL_MBS.MBS_Ref_Taster_DK_Pos_Foerderband,
    TON_PowerOnDelay_Compressor := PowerOnDelay_Compressor,
    TON_PowerOnDelay_Valve := PowerOnDelay_Valve_HorizontalMove,
    AutomaticMode := MBS_OperatingModes.F1
);
DmPD_Compressor_HorizontalMove := MBS_Skill_DmPB_PushWorkpieceOff.DO_ControlCompressorDmPD_01;
MBS_Skill_MR02_CuttingProcess(ESS := ((GVL.diNotAus_Kanal_A) AND (GVL.diNotAus_Kanal_B)), TouchSensor_01 := GVL_MBS.MBS_Ref_Taster_DK_Pos_Saege, AutomaticMode := MBS_OperatingModes.F1);
MR02_CuttingProcess := MBS_Skill_MR02_CuttingProcess.DO_CuttingProcessControlMR02;
MBS_Skill_CB_Moving(
    ESS := ((GVL.diNotAus_Kanal_A) AND (GVL.diNotAus_Kanal_B)),
    TouchSensor_01 := GVL_MBS.MBS_Ref_Taster_DK_Pos_Foerderband,
    LightSensor_01 := GVL_MBS.MBS_LS_Ende_Foerderband,
    TOF_Time_MotorControl := PowerOffDelay_ConveyorBelt,
    AutomaticMode := MBS_OperatingModes.F1
);
CB_MoveForwards := MBS_Skill_CB_Moving.DO_MovingHorizontalCB_01;

                
END_PROGRAM

PROGRAM SST_SkillSet
VAR
//Farbscanner- & Sortiertanlage Skills
	//ColorSensor Skills
	{attribute 'OPC.UA.DA':= '1'}
	SST_AutomaticColorDetection : SST_CS_AS_ColorDetection;
	
	//ConveyorBelt Skills
	{attribute 'OPC.UA.DA':= '1'}
	SST_ConveyorBeltMoveHorizontal_ToPD01 : SST_CB_AS_HorizontalMove;
	{attribute 'OPC.UA.DA':= '1'}
	SST_ConveyorBeltMoveHorizontal_ToPD02 : SST_CB_AS_HorizontalMove;
	{attribute 'OPC.UA.DA':= '1'}
	SST_ConveyorBeltMoveHorizontal_ToPD03 : SST_CB_AS_HorizontalMove;
	{attribute 'OPC.UA.DA':= '1'}
	SST_ConveyorBeltMoveHorizontal_TillEnd : SST_CB_AS_HorizontalMove;
	
	//PushingDeviceStation Skills
	{attribute 'OPC.UA.DA':= '1'}
	SST_PD01_HorizontalMove : SST_PD_AS_HorizontalMove;
	{attribute 'OPC.UA.DA':= '1'}
	SST_PD02_HorizontalMove : SST_PD_AS_HorizontalMove;
	{attribute 'OPC.UA.DA':= '1'}
	SST_PD03_HorizontalMove : SST_PD_AS_HorizontalMove;
	
	//Organisation FBs
	SST_OperatingModes : SST_OperatingModes;
	SST_ControlOfOutputs : SST_ControlOfOutputs;
	
	//InitialStateDrives	
	SST_PD_InitStateDrive: SST_PD_InitialStateDrive;

//Variablen zur Outputsteuerung
	//Output-Variablen der Komponente ConveyorBelt	
	CB_MoveForwardToPD01: BOOL;
	CB_MoveForwardToPD02: BOOL;
	CB_MoveForwardToPD03: BOOL;
	CB_MoveForwardTillEnd: BOOL;
	
	//Output-Variablen der Komponente PushingDevice
	PD01_Compressor : BOOL;
	PD02_Compressor : BOOL;
	PD03_Compressor : BOOL;
	PD01_Valve : BOOL;
	PD02_Valve : BOOL;
	PD03_Valve : BOOL;	
	
	//Output-Variablen für Init-Fahrt
	Init_PD01_Compressor : BOOL;
	Init_PD02_Compressor : BOOL;
	Init_PD03_Compressor : BOOL;
	Init_PD01_Valve : BOOL;
	Init_PD02_Valve : BOOL;
	Init_PD03_Valve : BOOL;
	
//Variablensetzung: Sollte später über SkillOA eingesetzt werden ODER Hard in SPS codiert (Diskussionspunkt)
	ResetButton: BOOL;
	StartButton: BOOL;
	ConfirmationButton: BOOL;

//Time Constraints
	TOF_Time_TransportPD01 : TIME;
	TOF_Time_TransportPD02 : TIME;
	TOF_Time_TransportPD03 : TIME;
	TON_Time_PD01Compressor : TIME;
	TON_Time_PD02Compressor : TIME;
	TON_Time_PD03Compressor : TIME;
	TON_Time_PD01Valve : TIME;
	TON_Time_PD02Valve : TIME;
	TON_Time_PD03Valve : TIME;
	TON_Time_PowerOFFSelfSet : TIME := T#150MS;
	
//Variable Values for InitialStateDrive
	MethodCall_InitStateDrive	: BOOL;
	InputVar_InitStateDrive		: BOOL;

END_VAR

                  SST_OperatingModes(
    Start := StartButton,
    Stop := ((GVL.diNotAus_Kanal_A) AND (GVL.diNotAus_Kanal_B)),
    Reset := ResetButton,
    Schalter := ConfirmationButton,
    Schrittkette_GS := (((SST_PD_InitStateDrive.ResetMethodCallMovePD01) AND (SST_PD_InitStateDrive.ResetMethodCallMovePD02) AND (SST_PD_InitStateDrive.ResetMethodCallMovePD03)))
);
SST_ControlOfOutputs(
    F4 := SST_OperatingModes.F4,
    F1 := SST_OperatingModes.F1,
    A2 := SST_OperatingModes.A2,
    A1 := SST_OperatingModes.A1,
    A6 := SST_OperatingModes.A6,
    Start := SST_OperatingModes.Start,
    CB_MoveForwardToPD01 := CB_MoveForwardToPD01,
    CB_MoveForwardToPD02 := CB_MoveForwardToPD02,
    CB_MoveForwardToPD03 := CB_MoveForwardToPD03,
    CB_MoveForwardTillEnd := CB_MoveForwardTillEnd,
    PD01_Compressor := PD01_Compressor,
    PD02_Compressor := PD02_Compressor,
    PD03_Compressor := PD03_Compressor,
    PD01_Valve := PD01_Valve,
    PD02_Valve := PD02_Valve,
    PD03_Valve := PD03_Valve,
    Init_PD01_Compressor := Init_PD01_Compressor,
    Init_PD02_Compressor := Init_PD02_Compressor,
    Init_PD03_Compressor := Init_PD03_Compressor,
    Init_PD01_Valve := Init_PD01_Valve,
    Init_PD02_Valve := Init_PD02_Valve,
    Init_PD03_Valve := Init_PD03_Valve
);
GVL_SST.SST_MOT_Foerderband := SST_ControlOfOutputs.ConveyorBeltForward;
SST_PD_InitStateDrive(
    MethodCall_InitDrive := MethodCall_InitStateDrive,
    ESS := ((GVL.diNotAus_Kanal_A) AND (GVL.diNotAus_Kanal_B)),
    InputInitialStateDrive := InputVar_InitStateDrive,
    TON_Time_PowerOFFSelfSet := TON_Time_PowerOFFSelfSet,
    InitDriveMode := SST_OperatingModes.A6
);
Init_PD01_Compressor := SST_PD_InitStateDrive.MotorControl_PD01_Compressor;
SST_AutomaticColorDetection(Color_Sensor := );
 := SST_AutomaticColorDetection.Color_White;
SST_ConveyorBeltMoveHorizontal_ToPD01(
    ESS := ((GVL.diNotAus_Kanal_A) AND (GVL.diNotAus_Kanal_B)),
    LightSensor_01 := GVL_SST.SST_LS_Eingang,
    LightSensor_02 := GVL_SST.SST_LS_nach_Farbsensor,
    TOF_Time_Motoransteuerung := TOF_Time_TransportPD01,
    AutomaticMode := SST_OperatingModes.A6
);
CB_MoveForwardToPD01 := SST_ConveyorBeltMoveHorizontal_ToPD01.DO_MovingConveyorBelt;
SST_ConveyorBeltMoveHorizontal_ToPD02(
    ESS := ((GVL.diNotAus_Kanal_A) AND (GVL.diNotAus_Kanal_B)),
    LightSensor_01 := GVL_SST.SST_LS_Eingang,
    LightSensor_02 := GVL_SST.SST_LS_nach_Farbsensor,
    TOF_Time_Motoransteuerung := TOF_Time_TransportPD02,
    AutomaticMode := SST_OperatingModes.A6
);
CB_MoveForwardToPD02 := SST_ConveyorBeltMoveHorizontal_ToPD02.DO_MovingConveyorBelt;
SST_ConveyorBeltMoveHorizontal_ToPD03(
    ESS := ((GVL.diNotAus_Kanal_A) AND (GVL.diNotAus_Kanal_B)),
    LightSensor_01 := GVL_SST.SST_LS_Eingang,
    LightSensor_02 := GVL_SST.SST_LS_nach_Farbsensor,
    TOF_Time_Motoransteuerung := TOF_Time_TransportPD03,
    AutomaticMode := SST_OperatingModes.A6
);
CB_MoveForwardToPD03 := SST_ConveyorBeltMoveHorizontal_ToPD03.DO_MovingConveyorBelt;
SST_ConveyorBeltMoveHorizontal_TillEnd(
    ESS := ((GVL.diNotAus_Kanal_A) AND (GVL.diNotAus_Kanal_B)),
    LightSensor_01 := GVL_SST.SST_LS_Eingang,
    LightSensor_02 := GVL_SST.SST_LS_nach_Farbsensor,
    TOF_Time_Motoransteuerung := ,
    AutomaticMode := SST_OperatingModes.A6
);
CB_MoveForwardTillEnd := SST_ConveyorBeltMoveHorizontal_TillEnd.DO_MovingConveyorBelt;
SST_PD01_HorizontalMove(
    ESS := ((GVL.diNotAus_Kanal_A) AND (GVL.diNotAus_Kanal_B)),
    LightSensor_01 := GVL_SST.SST_LS_nach_Farbsensor,
    LightSensor_02 := GVL_SST.SST_LS_weiss,
    PowerOnDelay_Compressor := TON_Time_PD01Compressor,
    PowerOnDelay_Valve := TON_Time_PD01Valve,
    AutomaticMode := SST_OperatingModes.A6
);
PD01_Compressor := SST_PD01_HorizontalMove.DO_ControlCompressorPD_01;
SST_PD02_HorizontalMove(
    ESS := ((GVL.diNotAus_Kanal_A) AND (GVL.diNotAus_Kanal_B)),
    LightSensor_01 := GVL_SST.SST_LS_nach_Farbsensor,
    LightSensor_02 := GVL_SST.SST_LS_rot,
    PowerOnDelay_Compressor := TON_Time_PD02Compressor,
    PowerOnDelay_Valve := TON_Time_PD02Valve,
    AutomaticMode := SST_OperatingModes.A6
);
PD02_Compressor := SST_PD02_HorizontalMove.DO_ControlCompressorPD_01;
SST_PD03_HorizontalMove(
    ESS := ((GVL.diNotAus_Kanal_A) AND (GVL.diNotAus_Kanal_B)),
    LightSensor_01 := GVL_SST.SST_LS_nach_Farbsensor,
    LightSensor_02 := GVL_SST.SST_LS_blau,
    PowerOnDelay_Compressor := TON_Time_PD03Compressor,
    PowerOnDelay_Valve := TON_Time_PD03Valve,
    AutomaticMode := SST_OperatingModes.A6
);
PD03_Compressor := SST_PD03_HorizontalMove.DO_ControlCompressorPD_01;

                
END_PROGRAM

PROGRAM VSG_SkillSet
VAR
    {attribute 'OPC.UA.DA':= '1'}
    VSG_ErrorDetected : BOOL := FALSE;

    {attribute 'OPC.UA.DA':= '1'}
    VSG_ErrorCode : UDINT := 0;

    {attribute 'OPC.UA.DA':= '1'}
    VSG_Skill_HorizontalMoveForwards : VSG_AS_HorizontalMoveEncoder;

    {attribute 'OPC.UA.DA':= '1'}
    VSG_Skill_HorizontalMoveBackwards : VSG_AS_HorizontalMoveEncoder;

    {attribute 'OPC.UA.DA':= '1'}
    VSG_Skill_VerticalMoveForwards : VSG_AS_VerticalMoveEncoder;

    {attribute 'OPC.UA.DA':= '1'}
    VSG_Skill_VerticalMoveBackwards : VSG_AS_VerticalMoveEncoder;

    {attribute 'OPC.UA.DA':= '1'}
    VSG_Skill_RotationMoveCW : VSG_AS_RotationMoveEncoder;

    {attribute 'OPC.UA.DA':= '1'}
    VSG_Skill_RotationMoveCCW : VSG_AS_RotationMoveEncoder;

    {attribute 'OPC.UA.DA':= '1'}
    VSG_Skill_SuctionProcess : VSG_AS_CompressorControl;

    VSG_ControlOfOutputs : VSG_ControlOfOutputs;
    VSG_OperatingModes : VSG_OperatingModes;
    VSG_DiagnosisHandler : VSG_DiagnosisHandler;
    VSG_InitialStateDrive : VSG_InitialStateDrive;
    bSuctionTrackingLatched : BOOL := FALSE;

    VSG_MoveHorizontalForwards01 : BOOL;
    VSG_MoveHorizontalForwards02 : BOOL;
    VSG_MoveHorizontalBackwards01 : BOOL;
    VSG_MoveHorizontalBackwards02 : BOOL;

    VSG_MoveVerticalDown01 : BOOL;
    VSG_MoveVerticalDown02 : BOOL;
    VSG_MoveVerticalUp01 : BOOL;
    VSG_MoveVerticalUp02 : BOOL;

    VSG_MoveRotationCW01 : BOOL;
    VSG_MoveRotationCW02 : BOOL;
    VSG_MoveRotationCCW01 : BOOL;
    VSG_MoveRotationCCW02 : BOOL;

    VSG_Compressor : BOOL;
    VSG_Valve : BOOL;

    Init_VSG_VertikalUp : BOOL;
    Init_VSG_VertikalDown : BOOL;
    Init_VSG_HorizontalForwards : BOOL;
    Init_VSG_HorizontalBackwards : BOOL;
    Init_VSG_RotationCW : BOOL;
    Init_VSG_RotationCCW : BOOL;

    ResetButton : BOOL;
    StartButton : BOOL;
    ConfirmationButton : BOOL;

    TIME_TSR : TIME := T#150MS;

    MethodCall_InitStateDrive : BOOL;
    InputVar_InitStateDrive : BOOL;
	sCurrentGemmaState: STRING(80);
	sLastNonFailureGemmaState : STRING(80) := '';
    rtD2 : R_TRIG;
END_VAR

                  IF GVL_Sim.bSimMode THEN

    GVL.diNotAus_Kanal_A := GVL_Sim.diNotAus_Kanal_A;
    GVL.diNotAus_Kanal_B := GVL_Sim.diNotAus_Kanal_B;

    GVL_VSG.VSG_Enc_vertikal_I1 := GVL_VSG_Sim.VSG_Enc_vertikal_I1;
    GVL_VSG.VSG_Enc_vertikal_I2 := GVL_VSG_Sim.VSG_Enc_vertikal_I2;

    GVL_VSG.VSG_Enc_horizontal_I1 := GVL_VSG_Sim.VSG_Enc_horizontal_I1;
    GVL_VSG.VSG_Enc_horizontal_I2 := GVL_VSG_Sim.VSG_Enc_horizontal_I2;

    GVL_VSG.VSG_Enc_drehen_I1 := GVL_VSG_Sim.VSG_Enc_drehen_I1;
    GVL_VSG.VSG_Enc_drehen_I2 := GVL_VSG_Sim.VSG_Enc_drehen_I2;

    GVL_VSG.VSG_Ref_Schalter_vertikal := GVL_VSG_Sim.VSG_Ref_Schalter_vertikal;
    GVL_VSG.VSG_Ref_Schalter_horizontal := GVL_VSG_Sim.VSG_Ref_Schalter_horizontal;
    GVL_VSG.VSG_Ref_Schalter_drehen := GVL_VSG_Sim.VSG_Ref_Schalter_drehen;

END_IF;


VSG_OperatingModes(
    Start := StartButton,
    Stop := NOT ((GVL.diNotAus_Kanal_A) AND (GVL.diNotAus_Kanal_B)),
    Reset := ResetButton,
    Schalter := ConfirmationButton,

    Schrittkette_GS :=
        VSG_InitialStateDrive.ResetMethodCall_RGB_Horizontal
        AND VSG_InitialStateDrive.ResetMethodCall_RGB_Vertical
        AND VSG_InitialStateDrive.ResetMethodCall_RotateCW,

    Count1 := 0,
    Count2 := 0,

    Alt_abort := OPCUA.Alt_abort,
    Err_detected := VSG_DiagnosisHandler.Err_detected,
    Diag_finished := VSG_DiagnosisHandler.Diag_finished,
    Alt_found := VSG_DiagnosisHandler.Alt_found,
    Cycle_finished := OPCUA.Cycle_finished
);


VSG_InitialStateDrive(
    MethodCall_InitDrive := MethodCall_InitStateDrive,
    ESS := ((GVL.diNotAus_Kanal_A) AND (GVL.diNotAus_Kanal_B)),
    InputInitDriveMode := InputVar_InitStateDrive,
    TouchSensor01_Rotation := GVL_VSG.VSG_Ref_Schalter_drehen,
    TouchSensor02_Vertical := GVL_VSG.VSG_Ref_Schalter_vertikal,
    TouchSensor03_horizontal := GVL_VSG.VSG_Ref_Schalter_horizontal,
    TOF_Time_TSR := TIME_TSR,
    InitDriveMode := VSG_OperatingModes.A6
);

Init_VSG_RotationCW := VSG_InitialStateDrive.VSG_Init_RotateCW;
Init_VSG_VertikalUp := VSG_InitialStateDrive.VSG_Init_VerticalUp;
Init_VSG_HorizontalBackwards := VSG_InitialStateDrive.VSG_Init_HorizontalBackwards;


VSG_Skill_HorizontalMoveForwards(
    ESS := ((GVL.diNotAus_Kanal_A) AND (GVL.diNotAus_Kanal_B)),
    TouchSensor01 := GVL_VSG.VSG_Ref_Schalter_horizontal,
    EncoderStartPosition01 := GVL_VSG.VSG_Enc_horizontal_I1,
    EncoderStartPosition02 := GVL_VSG.VSG_Enc_horizontal_I2,
    TOF_Time_TSR := TIME_TSR,
    AutomaticMode := VSG_OperatingModes.A6
);

VSG_MoveHorizontalForwards01 := VSG_Skill_HorizontalMoveForwards.DO_MovingHorizontalVSG_01;


VSG_Skill_HorizontalMoveBackwards(
    ESS := ((GVL.diNotAus_Kanal_A) AND (GVL.diNotAus_Kanal_B)),
    TouchSensor01 := GVL_VSG.VSG_Ref_Schalter_horizontal,
    EncoderStartPosition01 := GVL_VSG.VSG_Enc_horizontal_I1,
    EncoderStartPosition02 := GVL_VSG.VSG_Enc_horizontal_I2,
    TOF_Time_TSR := TIME_TSR,
    AutomaticMode := VSG_OperatingModes.A6
);

VSG_MoveHorizontalBackwards02 := VSG_Skill_HorizontalMoveBackwards.DO_MovingHorizontalVSG_01;


VSG_Skill_VerticalMoveForwards(
    ESS := ((GVL.diNotAus_Kanal_A) AND (GVL.diNotAus_Kanal_B)),
    TouchSensor01 := GVL_VSG.VSG_Ref_Schalter_vertikal,
    EncoderStartPosition01 := GVL_VSG.VSG_Enc_vertikal_I1,
    EncoderStartPosition02 := GVL_VSG.VSG_Enc_vertikal_I2,
    TOF_Time_TSR := TIME_TSR,
    AutomaticMode := VSG_OperatingModes.A6
);

VSG_MoveVerticalDown01 := VSG_Skill_VerticalMoveForwards.DO_MovingVerticalVSG_01;


VSG_Skill_VerticalMoveBackwards(
    ESS := ((GVL.diNotAus_Kanal_A) AND (GVL.diNotAus_Kanal_B)),
    TouchSensor01 := GVL_VSG.VSG_Ref_Schalter_vertikal,
    EncoderStartPosition01 := GVL_VSG.VSG_Enc_vertikal_I1,
    EncoderStartPosition02 := GVL_VSG.VSG_Enc_vertikal_I2,
    TOF_Time_TSR := TIME_TSR,
    AutomaticMode := VSG_OperatingModes.A6
);

VSG_MoveVerticalUp02 := VSG_Skill_VerticalMoveBackwards.DO_MovingVerticalVSG_01;


VSG_Skill_RotationMoveCW(
    ESS := ((GVL.diNotAus_Kanal_A) AND (GVL.diNotAus_Kanal_B)),
    TouchSensor01 := GVL_VSG.VSG_Ref_Schalter_drehen,
    EncoderStartPosition01 := GVL_VSG.VSG_Enc_drehen_I1,
    EncoderStartPosition02 := GVL_VSG.VSG_Enc_drehen_I2,
    TOF_Time_TSR := TIME_TSR,
    AutomaticMode := VSG_OperatingModes.A6
);

VSG_MoveRotationCW01 := VSG_Skill_RotationMoveCW.DO_MovingRotationVSG_01;


VSG_Skill_RotationMoveCCW(
    ESS := ((GVL.diNotAus_Kanal_A) AND (GVL.diNotAus_Kanal_B)),
    TouchSensor01 := GVL_VSG.VSG_Ref_Schalter_drehen,
    EncoderStartPosition01 := GVL_VSG.VSG_Enc_drehen_I1,
    EncoderStartPosition02 := GVL_VSG.VSG_Enc_drehen_I2,
    TOF_Time_TSR := TIME_TSR,
    AutomaticMode := VSG_OperatingModes.A6
);

VSG_MoveRotationCCW02 := VSG_Skill_RotationMoveCCW.DO_MovingRotationVSG_01;


VSG_Skill_SuctionProcess(
    ESS := ((GVL.diNotAus_Kanal_A) AND (GVL.diNotAus_Kanal_B)),

    EncoderStartPosition01 := GVL_VSG.VSG_Enc_drehen_I1,
    EncoderStartPosition02 := GVL_VSG.VSG_Enc_drehen_I2,
    EncoderStartPosition03 := GVL_VSG.VSG_Enc_horizontal_I1,
    EncoderStartPosition04 := GVL_VSG.VSG_Enc_horizontal_I2,
    EncoderStartPosition05 := GVL_VSG.VSG_Enc_vertikal_I1,
    EncoderStartPosition06 := GVL_VSG.VSG_Enc_vertikal_I2,

    WorkpieceAtPickupPosition := GVL_HRL.HRL_LS_aussen,

    AutomaticMode := VSG_OperatingModes.F1 AND NOT VSG_OperatingModes.D2
);

VSG_Compressor := VSG_Skill_SuctionProcess.DO_CompressorVSG;
VSG_Valve := VSG_Skill_SuctionProcess.DO_ValveVSG;

VSG_ErrorDetected := VSG_Skill_SuctionProcess.VSG_ErrorDetected;
VSG_ErrorCode := VSG_Skill_SuctionProcess.VSG_ErrorCode;


VSG_DiagnosisHandler(
    Diagnose_gefordert := VSG_OperatingModes.D2,
    ErrorDetectedRaw := VSG_Skill_SuctionProcess.VSG_ErrorDetected,
    Reset := ResetButton
);


VSG_ControlOfOutputs(
    F4 := VSG_OperatingModes.F4,
    F1 := VSG_OperatingModes.F1,
    A2 := VSG_OperatingModes.A2,
    A1 := VSG_OperatingModes.A1,
    A6 := VSG_OperatingModes.A6,
    Start := VSG_OperatingModes.Start,

    VSG_VertikalDown01 := VSG_MoveVerticalDown01,
    VSG_VertikalDown02 := VSG_MoveVerticalDown02,
    VSG_VertikalUp01 := VSG_MoveVerticalUp01,
    VSG_VertikalUp02 := VSG_MoveVerticalUp02,

    VSG_HorizontalForwards01 := VSG_MoveHorizontalForwards01,
    VSG_HorizontalForwards02 := VSG_MoveHorizontalForwards02,
    VSG_HorizontalBackwards01 := VSG_MoveHorizontalBackwards01,
    VSG_HorizontalBackwards02 := VSG_MoveHorizontalBackwards02,

    VSG_RotationCW01 := VSG_MoveRotationCW01,
    VSG_RotationCW02 := VSG_MoveRotationCW02,
    VSG_RotationCCW01 := VSG_MoveRotationCCW01,
    VSG_RotationCCW02 := VSG_MoveRotationCCW02,

    VSG_Compressor := VSG_Compressor,
    VSG_Valve := VSG_Valve,

    Init_VSG_VertikalUp := Init_VSG_VertikalUp,
    Init_VSG_VertikalDown := Init_VSG_VertikalDown,
    Init_VSG_HorizontalForwards := Init_VSG_HorizontalForwards,
    Init_VSG_HorizontalBackwards := Init_VSG_HorizontalBackwards,
    Init_VSG_RotationCW := Init_VSG_RotationCW,
    Init_VSG_RotationCCW := Init_VSG_RotationCCW
);


IF GVL_Sim.bSimMode THEN

    GVL_VSG_Sim.VSG_MOT_vertikal_runter := VSG_ControlOfOutputs.MoveVerticalDown;
    GVL_VSG_Sim.VSG_MOT_vertikal_hoch := VSG_ControlOfOutputs.MoveVerticalUp;

    GVL_VSG_Sim.VSG_MOT_horizontal_vorwaerts := VSG_ControlOfOutputs.MoveHorizontalForwards;
    GVL_VSG_Sim.VSG_MOT_horizontal_rueckwaerts := VSG_ControlOfOutputs.MoveHorizontalBackwards;

    GVL_VSG_Sim.VSG_MOT_drehen_CW := VSG_ControlOfOutputs.MoveRotationCW;
    GVL_VSG_Sim.VSG_MOT_drehen_CCW := VSG_ControlOfOutputs.MoveRotationCCW;

    GVL_VSG_Sim.VSG_Kompressor := VSG_ControlOfOutputs.CompressorON;
    GVL_VSG_Sim.VSG_MV_Vakuum := VSG_ControlOfOutputs.ValveON;

ELSE

    GVL_VSG.VSG_MOT_vertikal_runter := VSG_ControlOfOutputs.MoveVerticalDown;
    GVL_VSG.VSG_MOT_vertikal_hoch := VSG_ControlOfOutputs.MoveVerticalUp;

    GVL_VSG.VSG_MOT_horizontal_vorwaerts := VSG_ControlOfOutputs.MoveHorizontalForwards;
    GVL_VSG.VSG_MOT_horizontal_rueckwaerts := VSG_ControlOfOutputs.MoveHorizontalBackwards;

    GVL_VSG.VSG_MOT_drehen_CW := VSG_ControlOfOutputs.MoveRotationCW;
    GVL_VSG.VSG_MOT_drehen_CCW := VSG_ControlOfOutputs.MoveRotationCCW;

    GVL_VSG.VSG_Kompressor := VSG_ControlOfOutputs.CompressorON;
    GVL_VSG.VSG_MV_Vakuum := VSG_ControlOfOutputs.ValveON;

END_IF;

//GEMMA_Mappings
IF VSG_OperatingModes.A1 THEN
    sCurrentGemmaState := 'VSG_OperatingModes.A1';
ELSIF VSG_OperatingModes.A2 THEN
    sCurrentGemmaState := 'VSG_OperatingModes.A2';
ELSIF VSG_OperatingModes.A5 THEN
    sCurrentGemmaState := 'VSG_OperatingModes.A5';
ELSIF VSG_OperatingModes.A6 THEN
    sCurrentGemmaState := 'VSG_OperatingModes.A6';
ELSIF VSG_OperatingModes.F1 THEN
    sCurrentGemmaState := 'VSG_OperatingModes.F1';
ELSIF VSG_OperatingModes.F4 THEN
    sCurrentGemmaState := 'VSG_OperatingModes.F4';
ELSIF VSG_OperatingModes.D1 THEN
    sCurrentGemmaState := 'VSG_OperatingModes.D1';
ELSIF VSG_OperatingModes.D3 THEN
    sCurrentGemmaState := 'VSG_OperatingModes.D3';
END_IF;

IF NOT VSG_OperatingModes.D2 THEN
    sLastNonFailureGemmaState := sCurrentGemmaState;
END_IF;

rtD2(CLK := VSG_OperatingModes.D2);

IF rtD2.Q THEN
    OPCUA.LastGEMMAStateBeforeFailure := sLastNonFailureGemmaState;
END_IF;
                
END_PROGRAM

FUNCTION_BLOCK AutomaticColorDetection_nichtfertig
VAR_INPUT
	MethodCall : BOOL;
	EmergencyStopSignal : BOOL;
	ColorSensor: INT;
	ColorCode_1: INT;
	ColorCode_2: INT;
	ColorCode_3: INT;
	OperatingMode : BOOL;
END_VAR

VAR_OUTPUT
	Color_1: BOOL;
	Color_2: BOOL;
	Color_3: BOOL;
END_VAR

VAR
END_VAR

                  Color_1 := ((ColorSensor) = (ColorCode_1));
Color_2 := ((ColorSensor) = (ColorCode_2));
Color_3 := ((ColorSensor) = (Color_3));
                
END_FUNCTION_BLOCK

FUNCTION_BLOCK AxisControl_Encoder
VAR_INPUT //Input-Variablen des FBs
	MethodCall					: BOOL; // Variable zum aktiven Aufruf einer OPC UA Methode
	EmergencyStopSignal 		: BOOL; // Variable für Not-Signal 
	Direction 					: BOOL; // Variable zur Bestimmung der Bewegungsrichtung
	InitStateDrive_Input		: BOOL; //InputVariable für Initialfahrt
	DI01 						: BOOL; // Digitaler Input wie bspw. Lichtsensor oder Kontaktsensor 
	DI02_EncoderStart01			: UDINT; // Digitaler Input Encoder Wert
	DI03_EncoderTarget01		: UDINT; // Digitaler Input Encoder Wert
	DI04_EncoderStart02			: UDINT; // Digitaler Input Encoder Wert
	DI05_EncoderTarget02		: UDINT; // Digitaler Input Encoder Wert
	TouchSensorRelief 			: BOOL; // Hilfsvariable zur Identifikation ob eine Endschalterentlastung notwendig ist
	TOF_Time_MotorControl		: TIME; // Zeitvariable für die Ausschaltverzögerung des digitalen Outputs (Motoransteuerung) 
	TOF_Time_TouchSensorRelief	: TIME; // Ausschaltverzögerung für die Endschaltentlastung
	OperatingMode				: BOOL; // Variable zur Festlegung des benötigten Betriebszustandes für die Auslösung des FBs
END_VAR

VAR_OUTPUT //Output-Variablen des FBs
	DigitalOutputControl_01	: BOOL; //Digitale Output Ansteuerung des Motor 1
	DigitalOutputControl_02	: BOOL; //Digitale Output Ansteuerung des Motor 2
	ResetMethodCall			: BOOL; //Outputvariable für den Reset der OPC UA Methode
END_VAR

VAR //Interne-Variablen des FBs
//FlipFlop
	RS_AxisControl		: RS; //FlipFlop für die Ansteuerung der Achse oder des Transportbandes
	RS_TouchSensorRelief: RS; //FlipFlop zu Ansteuerung der Endschalterentlastung
//Zeitverzögerung
	TOF_TouchSensorRelief	: TOF; //Ausschaltverzögerung für die Endschalterentlastung
	TOF_DigitalOutputControl: TOF; //Ausschaltverzögerung für die Outputansteuerung
//Flanke	
	R_TRIG_MethodCall			: R_TRIG; //Flankenerkennung für eingehenden MethodenCall
	R_TRIG_EncoderPos01_Input	: R_TRIG; //Flankenerkennung für Vergleich der Encoderwerte von Start- und Zielposition
	R_TRIG_EncoderPos02_Input	: R_TRIG; //Flankenerkennung für Vergleich der Encoderwerte von Start- und Zielposition
	R_TRIG_EncoderPos01_Output	: R_TRIG; //Flankenerkennung für Vergleich der Encoderwerte von Start- und Zielposition
	R_TRIG_EncoderPos02_Output	: R_TRIG; //Flankenerkennung für Vergleich der Encoderwerte von Start- und Zielposition
END_VAR

                  R_TRIG_MethodCall(CLK := MethodCall);

ResetMethodCall := (
    (Direction AND (DI02_EncoderStart01 >= DI03_EncoderTarget01) AND (DI04_EncoderStart02 >= DI05_EncoderTarget02))
    OR ((NOT Direction) AND (DI02_EncoderStart01 <= DI03_EncoderTarget01) AND (DI04_EncoderStart02 <= DI05_EncoderTarget02))
    OR EmergencyStopSignal
    OR DI01
    OR InitStateDrive_Input
);

RS_AxisControl(
    SET := (
        R_TRIG_MethodCall.Q
        AND (
            (Direction AND (DI02_EncoderStart01 < DI03_EncoderTarget01) AND (DI04_EncoderStart02 < DI05_EncoderTarget02))
            OR ((NOT Direction) AND (DI02_EncoderStart01 > DI03_EncoderTarget01) AND (DI04_EncoderStart02 > DI05_EncoderTarget02))
            OR InitStateDrive_Input
        )
        AND OperatingMode
    ),
    RESET1 := ResetMethodCall
);

TOF_DigitalOutputControl(IN := RS_AxisControl.Q1, PT := TOF_Time_MotorControl);
DigitalOutputControl_01 := TOF_DigitalOutputControl.Q;

RS_TouchSensorRelief(
    SET := ((ResetMethodCall) AND (MethodCall) AND (TouchSensorRelief)),
    RESET1 := ((NOT DI01) OR EmergencyStopSignal OR InitStateDrive_Input)
);
TOF_TouchSensorRelief(IN := RS_TouchSensorRelief.Q1, PT := TOF_Time_TouchSensorRelief);
DigitalOutputControl_02 := TOF_TouchSensorRelief.Q;

                
END_FUNCTION_BLOCK

FUNCTION_BLOCK AxisControl_MultipleInputSensors
VAR_INPUT//Input-Variablen des FBs
	MethodCall					: BOOL; // Variable zum aktiven Aufruf einer OPC UA Methode
	EmergencyStopSignal 		: BOOL; // Variable für Not-Signal 
	Direction 					: BOOL; // Variable zur Bestimmung der Bewegungsrichtung
	InitStateDrive_Input		: BOOL; //InputVariable für Initialfahrt
	DI01 						: BOOL; // Digitaler Input wie bspw. Lichtsensor oder Kontaktsensor 
	DI02 						: BOOL; // Digitaler Input wie bspw. Lichtsensor oder Kontaktsensor 
	TouchSensorRelief			: BOOL; // Hilfsvariable zur Identifikation ob eine Endschalterentlastung notwendig ist
	TOF_Time_MotorControl		: TIME; // Zeitvariable für die Ausschaltverzögerung des digitalen Outputs (Motoransteuerung) 
	TOF_Time_TouchSensorRelief	: TIME; // Ausschaltverzögerung für die Endschaltentlastung
	OperatingMode				: BOOL; // Variable zur Festlegung des benötigten Betriebszustandes für die Auslösung des FBs
END_VAR

VAR_OUTPUT //Output-Variablen des FBs
	DigitalOutputControl_01	: BOOL; //Digitale Output Ansteuerung des Motor 1
	DigitalOutputControl_02	: BOOL; //Digitale Output Ansteuerung des Motor 2
	ResetMethodCall			: BOOL; //Outputvariable für den Reset der OPC UA Methode
	InitStateDriveFinished	: BOOL;
	Count1 : INT := 0;
	Count2 : INT := 0;
END_VAR

VAR //Interne-Variablen des FBs
//FlipFlop
	RS_AxisControl		: RS; //FlipFlop für die Ansteuerung der Achse oder des Transportbandes
	RS_TouchSensorRelief: RS; //FlipFlop zu Ansteuerung der Endschalterentlastung
//Zeitverzögerung
	TOF_TouchSensorRelief	: TOF; //Ausschaltverzögerung für die Endschalterentlastung
	TOF_DigitalOutputControl: TOF; //Ausschaltverzögerung für die Outputansteuerung	
//Flanke	
	R_TRIG_MethodCall : R_TRIG; //Flankenerkennung für eingehenden MethodenCall
	R_TRIG_TSR : R_TRIG; //Flankenerkennung für eingehenden MethodenCall
	F_TRIG_0: F_TRIG;
	F_TRIG_1: F_TRIG;
END_VAR

                  R_TRIG_MethodCall(CLK := MethodCall);
ResetMethodCall := ((((Direction) AND (DI02))) OR (EmergencyStopSignal));
RS_AxisControl(
    SET := ((R_TRIG_MethodCall.Q) AND (((((Direction) AND (((DI01) OR (TouchSensorRelief))))) OR (((Direction) AND (InitStateDrive_Input))))) AND (OperatingMode)),
    RESET1 := ((((Direction) AND (DI02))) OR (EmergencyStopSignal))
);
TOF_DigitalOutputControl(IN := RS_AxisControl.Q1, PT := TOF_Time_MotorControl);
DigitalOutputControl_01 := TOF_DigitalOutputControl.Q;
R_TRIG_TSR(CLK := ((ResetMethodCall) AND (DI02) AND (MethodCall) AND (TouchSensorRelief)));
InitStateDriveFinished := ((NOT (DI02)) OR (EmergencyStopSignal));
RS_TouchSensorRelief(SET := R_TRIG_TSR.Q, RESET1 := ((NOT (DI02)) OR (EmergencyStopSignal)));
TOF_TouchSensorRelief(IN := RS_TouchSensorRelief.Q1, PT := TOF_Time_TouchSensorRelief);
DigitalOutputControl_02 := TOF_TouchSensorRelief.Q;
F_TRIG_0(CLK := DigitalOutputControl_01);
F_TRIG_1(CLK := DigitalOutputControl_02);

                
END_FUNCTION_BLOCK

FUNCTION_BLOCK CompressorControl
VAR_INPUT
    MethodCall : BOOL;
    EmergencyStopSignal : BOOL;
    Destination : BOOL;
    InitStateDrive_Input : BOOL;

    DI01 : BOOL;
    DI02 : BOOL;

    DI03_EncoderStart01 : UDINT;
    DI04_EncoderStart02 : UDINT;
    DI05_EncoderStart03 : UDINT;
    DI06_EncoderStart04 : UDINT;
    DI07_EncoderStart05 : UDINT;
    DI08_EncoderStart06 : UDINT;

    DI09_EncoderTarget01 : UDINT;
    DI10_EncoderTarget02 : UDINT;
    DI11_EncoderTarget03 : UDINT;
    DI12_EncoderTarget04 : UDINT;
    DI13_EncoderTarget05 : UDINT;
    DI14_EncoderTarget06 : UDINT;

    PowerOFF_SelfSet : BOOL;
    TON_Time_PowerOFFSelfSet : TIME;
    TON_Time_Compressor : TIME;
    TON_Time_Valve : TIME;
    OperatingMode : BOOL;
END_VAR

VAR_OUTPUT
    DigitalOutputControl_01 : BOOL;
    DigitalOutputControl_02 : BOOL;
    ResetMethodCall : BOOL;
END_VAR

VAR
    RS_Compressor : RS;
    RS_Valve : RS;

    TON_Compressor_Control : TON;
    TON_Valve_Control : TON;
    TON_SelfSet : TON;

    R_TRIG_MethodCall : R_TRIG;

    R_TRIG_EncoderPos01_CompressorInput : R_TRIG;
    R_TRIG_EncoderPos02_CompressorInput : R_TRIG;
    R_TRIG_EncoderPos03_CompressorInput : R_TRIG;
    R_TRIG_EncoderPos04_CompressorInput : R_TRIG;
    R_TRIG_EncoderPos05_CompressorInput : R_TRIG;
    R_TRIG_EncoderPos06_CompressorInput : R_TRIG;

    R_TRIG_EncoderPos01_CompressorOutput : R_TRIG;
    R_TRIG_EncoderPos02_CompressorOutput : R_TRIG;
    R_TRIG_EncoderPos03_CompressorOutput : R_TRIG;
    R_TRIG_EncoderPos04_CompressorOutput : R_TRIG;
    R_TRIG_EncoderPos05_CompressorOutput : R_TRIG;
    R_TRIG_EncoderPos06_CompressorOutput : R_TRIG;

    R_TRIG_EncoderPos01_ValveInput : R_TRIG;
    R_TRIG_EncoderPos02_ValveInput : R_TRIG;
    R_TRIG_EncoderPos03_ValveInput : R_TRIG;
    R_TRIG_EncoderPos04_ValveInput : R_TRIG;
    R_TRIG_EncoderPos05_ValveInput : R_TRIG;
    R_TRIG_EncoderPos06_ValveInput : R_TRIG;

    R_TRIG_EncoderPos01_ValveOutput : R_TRIG;
    R_TRIG_EncoderPos02_ValveOutput : R_TRIG;
    R_TRIG_EncoderPos03_ValveOutput : R_TRIG;
    R_TRIG_EncoderPos04_ValveOutput : R_TRIG;
    R_TRIG_EncoderPos05_ValveOutput : R_TRIG;
    R_TRIG_EncoderPos06_ValveOutput : R_TRIG;

    bEncoderInputCondition : BOOL;
    bEncoderOutputCondition : BOOL;
    bStartCondition : BOOL;
    bResetCondition : BOOL;
END_VAR

                  R_TRIG_MethodCall(CLK := MethodCall);

R_TRIG_EncoderPos01_CompressorInput(CLK := DI03_EncoderStart01 <> DI09_EncoderTarget01);
R_TRIG_EncoderPos02_CompressorInput(CLK := DI04_EncoderStart02 <> DI10_EncoderTarget02);
R_TRIG_EncoderPos03_CompressorInput(CLK := DI05_EncoderStart03 <> DI11_EncoderTarget03);
R_TRIG_EncoderPos04_CompressorInput(CLK := DI06_EncoderStart04 <> DI12_EncoderTarget04);
R_TRIG_EncoderPos05_CompressorInput(CLK := DI07_EncoderStart05 <> DI13_EncoderTarget05);
R_TRIG_EncoderPos06_CompressorInput(CLK := DI08_EncoderStart06 <> DI14_EncoderTarget06);

R_TRIG_EncoderPos01_CompressorOutput(CLK := DI03_EncoderStart01 = DI09_EncoderTarget01);
R_TRIG_EncoderPos02_CompressorOutput(CLK := DI04_EncoderStart02 = DI10_EncoderTarget02);
R_TRIG_EncoderPos03_CompressorOutput(CLK := DI05_EncoderStart03 = DI11_EncoderTarget03);
R_TRIG_EncoderPos04_CompressorOutput(CLK := DI06_EncoderStart04 = DI12_EncoderTarget04);
R_TRIG_EncoderPos05_CompressorOutput(CLK := DI07_EncoderStart05 = DI13_EncoderTarget05);
R_TRIG_EncoderPos06_CompressorOutput(CLK := DI08_EncoderStart06 = DI14_EncoderTarget06);

R_TRIG_EncoderPos01_ValveInput(CLK := DI03_EncoderStart01 <> DI09_EncoderTarget01);
R_TRIG_EncoderPos02_ValveInput(CLK := DI04_EncoderStart02 <> DI10_EncoderTarget02);
R_TRIG_EncoderPos03_ValveInput(CLK := DI05_EncoderStart03 <> DI11_EncoderTarget03);
R_TRIG_EncoderPos04_ValveInput(CLK := DI06_EncoderStart04 <> DI12_EncoderTarget04);
R_TRIG_EncoderPos05_ValveInput(CLK := DI07_EncoderStart05 <> DI13_EncoderTarget05);
R_TRIG_EncoderPos06_ValveInput(CLK := DI08_EncoderStart06 <> DI14_EncoderTarget06);

R_TRIG_EncoderPos01_ValveOutput(CLK := DI03_EncoderStart01 = DI09_EncoderTarget01);
R_TRIG_EncoderPos02_ValveOutput(CLK := DI04_EncoderStart02 = DI10_EncoderTarget02);
R_TRIG_EncoderPos03_ValveOutput(CLK := DI05_EncoderStart03 = DI11_EncoderTarget03);
R_TRIG_EncoderPos04_ValveOutput(CLK := DI06_EncoderStart04 = DI12_EncoderTarget04);
R_TRIG_EncoderPos05_ValveOutput(CLK := DI07_EncoderStart05 = DI13_EncoderTarget05);
R_TRIG_EncoderPos06_ValveOutput(CLK := DI08_EncoderStart06 = DI14_EncoderTarget06);

bEncoderInputCondition :=
    R_TRIG_EncoderPos01_CompressorInput.Q
    AND R_TRIG_EncoderPos02_CompressorInput.Q
    AND R_TRIG_EncoderPos03_CompressorInput.Q
    AND R_TRIG_EncoderPos04_CompressorInput.Q
    AND R_TRIG_EncoderPos05_CompressorInput.Q
    AND R_TRIG_EncoderPos06_CompressorInput.Q;

bEncoderOutputCondition :=
    R_TRIG_EncoderPos01_CompressorOutput.Q
    AND R_TRIG_EncoderPos02_CompressorOutput.Q
    AND R_TRIG_EncoderPos03_CompressorOutput.Q
    AND R_TRIG_EncoderPos04_CompressorOutput.Q
    AND R_TRIG_EncoderPos05_CompressorOutput.Q
    AND R_TRIG_EncoderPos06_CompressorOutput.Q;

bStartCondition :=
    (DI01 OR bEncoderInputCondition OR InitStateDrive_Input)
    AND OperatingMode;

bResetCondition :=
    (Destination AND (DI02 OR bEncoderOutputCondition))
    OR EmergencyStopSignal;

ResetMethodCall := bResetCondition;

RS_Compressor(
    SET := R_TRIG_MethodCall.Q AND bStartCondition,
    RESET1 := bResetCondition
);

TON_Compressor_Control(
    IN := RS_Compressor.Q1,
    PT := TON_Time_Compressor
);

DigitalOutputControl_01 := TON_Compressor_Control.Q;

TON_SelfSet(
    IN := R_TRIG_MethodCall.Q AND PowerOFF_SelfSet,
    PT := TON_Time_PowerOFFSelfSet
);

RS_Valve(
    SET := R_TRIG_MethodCall.Q AND (DI01 OR bEncoderInputCondition OR InitStateDrive_Input),
    RESET1 := (Destination AND (DI02 OR bEncoderOutputCondition OR TON_SelfSet.Q)) OR EmergencyStopSignal
);

TON_Valve_Control(
    IN := RS_Valve.Q1,
    PT := TON_Time_Valve
);

DigitalOutputControl_02 := TON_Valve_Control.Q;
                
END_FUNCTION_BLOCK

FUNCTION_BLOCK CuttingProcess
VAR_INPUT//Input-Variablen des FBs
	MethodCall			: BOOL; // Variable zum aktiven Aufruf einer OPC UA Methode
	EmergencyStopSignal : BOOL; // Variable für Not-Signal
	InitStateDrive_Input: BOOL; //InputVariable für Initialfahrt
	DI01				: BOOL; // Digitaler Input wie bspw. Lichtsensor oder Kontaktsensor
	TOF_Time_CuttingTime: TIME; // Ausschaltverzögerung für die Rücksetzbedingung um eine Bearbeitungszeit zu simulieren
	OperatingMode		: BOOL; // Variable zur Festlegung des benötigten Betriebszustandes für die Auslösung des FBs
END_VAR

VAR_OUTPUT //Output-Variablen des FBs
	DigitalOutputControl_01	: BOOL; //Digitale Output Ansteuerung des Motor 1
	ResetMethodCall			: BOOL; //Outputvariable für den Reset der OPC UA Methode
END_VAR

VAR //Interne-Variablen des FBs
//FlipFlop
	RS_CuttingProcess: RS; //FlipFlop für die Ansteuerung der Schneidemaschine
//Zeitverzögerung
	TOF_CuttingTime: TOF; //Ausschaltverzögerung simulativ für die Bearbeitungszeit
//Flanke	
	R_TRIG_MethodCall: R_TRIG; //Flankenerkennung für eingehenden MethodenCall
END_VAR

                  R_TRIG_MethodCall(CLK := MethodCall);
R_TRIG_MethodCall(CLK := MethodCall);
TOF_CuttingTime(IN := R_TRIG_MethodCall.Q, PT := TOF_Time_CuttingTime);
ResetMethodCall := ((TOF_CuttingTime.Q) OR (EmergencyStopSignal));
RS_CuttingProcess(SET := ((R_TRIG_MethodCall.Q) AND (((DI01) OR (InitStateDrive_Input))) AND (OperatingMode)), RESET1 := ((TOF_CuttingTime.Q) OR (EmergencyStopSignal)));
DigitalOutputControl_01 := RS_CuttingProcess.Q1;
                
END_FUNCTION_BLOCK

FUNCTION_BLOCK HardeningProcess
VAR_INPUT//Input-Variablen des FBs
	MethodCall				: BOOL; // Variable zum aktiven Aufruf einer OPC UA Methode
	EmergencyStopSignal 	: BOOL; // Variable für Not-Signal
	InitStateDrive_Input	: BOOL; //InputVariable für Initialfahrt
	DI01					: BOOL; // Digitaler Input wie bspw. Lichtsensor oder Kontaktsensor
	TOF_Time_HardeningTime	: TIME; // Ausschaltverzögerung für die Rücksetzbedingung um eine Bearbeitungszeit zu simulieren
	OperatingMode			: BOOL; // Variable zur Festlegung des benötigten Betriebszustandes für die Auslösung des FBs
END_VAR

VAR_OUTPUT //Output-Variablen des FBs
	DigitalOutputControl_01	: BOOL; //Digitale Output Ansteuerung des Motor 1
	ResetMethodCall			: BOOL; //Outputvariable für den Reset der OPC UA Methode
END_VAR

VAR //Interne-Variablen des FBs
//FlipFlop
	RS_HardeningProcess: RS; //FlipFlop für die Ansteuerung des Ofens
//Zeitverzögerung
	TOF_HardeningTime: TOF; //Ausschaltverzögerung simulativ für die Bearbeitungszeit
//Flanke	
	R_TRIG_MethodCall: R_TRIG; //Flankenerkennung für eingehenden MethodenCall
END_VAR

                  R_TRIG_MethodCall(CLK := MethodCall);
R_TRIG_MethodCall(CLK := MethodCall);
TOF_HardeningTime(IN := R_TRIG_MethodCall.Q, PT := TOF_Time_HardeningTime);
ResetMethodCall := ((TOF_HardeningTime.Q) AND (EmergencyStopSignal));
RS_HardeningProcess(SET := ((R_TRIG_MethodCall.Q) AND (((DI01) OR (InitStateDrive_Input))) AND (OperatingMode)), RESET1 := ((TOF_HardeningTime.Q) AND (EmergencyStopSignal)));
DigitalOutputControl_01 := RS_HardeningProcess.Q1;
                
END_FUNCTION_BLOCK

FUNCTION_BLOCK SecuringWorkpiece
VAR_INPUT//Input-Variablen des FBs
	MethodCall				: BOOL; // Variable zum aktiven Aufruf einer OPC UA Methode
	EmergencyStopSignal 	: BOOL; // Variable für Not-Signal 
	InitStateDrive_Input	: BOOL; //InputVariable für Initialfahrt
	DI01 					: BOOL; // Digitaler Input wie bspw. Lichtsensor oder Kontaktsensor 
	TON_Time_Securing		: TIME;	// Einschaltverzögerung um eine Bearbeitungszeit zu simulieren
	TON_Time_SecuringProcess: TIME; // Einschaltverzögerung um einen Einspannprozess zu simulieren
	OperatingMode			: BOOL; // Variable zur Festlegung des benötigten Betriebszustandes für die Auslösung des FBs
END_VAR

VAR_OUTPUT //Output-Variablen des FBs
	DigitalOutputControl_01	: BOOL; //Digitale Output Ansteuerung des Motor 1
	DigitalOutputControl_02	: BOOL; //Digitale Output Ansteuerung des Motor 2
	ResetMethodCall			: BOOL; //Outputvariable für den Reset der OPC UA Methode
END_VAR

VAR //Interne-Variablen des FBs
//FlipFlop
	RS_SecuringProcessCompressorON	: RS; //FlipFlop für die Ansteuerung des Compressors
	RS_SecuringProcessCompressorOFF	: RS; //FlipFlop für die Ansteuerung des Ventils	
//Zeitverzögerung
	TON_SecuringTime_Compressor	: TON; //Einschaltverzögerung für Einspannzeit
	TON_SecuringTime_Valve		: TON; //Einschaltverzögerung für Einspannzeit
	TON_SecuringProcessingTime	: TON; //Einschaltverzögerung zur Simulation von einer Gesamtbearbeitungszeit
//Flanke	
	R_TRIG_MethodCall: R_TRIG; //Flankenerkennung für eingehenden MethodenCall
END_VAR

                  R_TRIG_MethodCall(CLK := MethodCall);
R_TRIG_MethodCall(CLK := MethodCall);
TON_SecuringProcessingTime(IN := R_TRIG_MethodCall.Q, PT := TON_Time_SecuringProcess);
RS_SecuringProcessCompressorON(SET := ((R_TRIG_MethodCall.Q) AND (((DI01) OR (InitStateDrive_Input))) AND (OperatingMode)), RESET1 := ((TON_SecuringProcessingTime.Q) OR (EmergencyStopSignal)));
TON_SecuringTime_Compressor(IN := RS_SecuringProcessCompressorON.Q1, PT := TON_Time_Securing);
DigitalOutputControl_01 := TON_SecuringTime_Compressor.Q;
R_TRIG_MethodCall(CLK := MethodCall);
R_TRIG_MethodCall(CLK := MethodCall);
TON_SecuringProcessingTime(IN := R_TRIG_MethodCall.Q, PT := TON_Time_SecuringProcess);
ResetMethodCall := ((TON_SecuringProcessingTime.Q) OR (EmergencyStopSignal));
RS_SecuringProcessCompressorOFF(SET := ((R_TRIG_MethodCall.Q) AND (((DI01) OR (InitStateDrive_Input))) AND (OperatingMode)), RESET1 := ((TON_SecuringProcessingTime.Q) OR (EmergencyStopSignal)));
TON_SecuringTime_Valve(IN := RS_SecuringProcessCompressorOFF.Q1, PT := TON_Time_Securing + T#0.5s);
DigitalOutputControl_02 := TON_SecuringTime_Valve.Q;

                
END_FUNCTION_BLOCK

FUNCTION_BLOCK StampingProcess
VAR_INPUT//Input-Variablen des FBs
	MethodCall				: BOOL; // Variable zum aktiven Aufruf einer OPC UA Methode
	EmergencyStopSignal 	: BOOL; // Variable für Not-Signal
	InitStateDrive_Input	: BOOL; //InputVariable für Initialfahrt
	DI01					: BOOL; // Digitaler Input wie bspw. Lichtsensor oder Kontaktsensor
	TOF_Time_StampingTime	: TIME; // Ausschaltverzögerung für die Rücksetzbedingung um eine Bearbeitungszeit zu simulieren
	OperatingMode			: BOOL; // Variable zur Festlegung des benötigten Betriebszustandes für die Auslösung des FBs
END_VAR

VAR_OUTPUT //Output-Variablen des FBs
	DigitalOutputControl_01	: BOOL; //Digitale Output Ansteuerung des Motor 1
	ResetMethodCall			: BOOL; //Outputvariable für den Reset der OPC UA Methode
END_VAR

VAR //Interne-Variablen des FBs
//FlipFlop
	RS_StampingProcess: RS; //FlipFlop für die Ansteuerung der Stanzmaschine
//Zeitverzögerung
	TOF_StampingTime: TOF; //Ausschaltverzögerung simulativ für die Bearbeitungszeit
//Flanke	
	R_TRIG_MethodCall: R_TRIG; //Flankenerkennung für eingehenden MethodenCall
END_VAR

                  
R_TRIG_MethodCall(CLK := MethodCall);
R_TRIG_MethodCall(CLK := MethodCall);
TOF_StampingTime(IN := R_TRIG_MethodCall.Q, PT := TOF_Time_StampingTime);
ResetMethodCall := ((TOF_StampingTime.Q) AND (EmergencyStopSignal));
RS_StampingProcess(SET := ((R_TRIG_MethodCall.Q) AND (((DI01) OR (InitStateDrive_Input))) AND (OperatingMode)), RESET1 := ((TOF_StampingTime.Q) AND (EmergencyStopSignal)));
DigitalOutputControl_01 := RS_StampingProcess.Q1;
                
END_FUNCTION_BLOCK

FUNCTION_BLOCK HRL_ControlOfOutputs
VAR_INPUT
	F4							: BOOL;
	F1							: BOOL;
	A2							: BOOL;
	A6							: BOOL;
	A1							: BOOL := FALSE;
	Start						: BOOL;
	CB_forwards 				: BOOL; 
	CB_backwards 				: BOOL; 
	RGB_Forwards01 				: BOOL;
	RGB_Forwards02 				: BOOL;
	RGB_Backwards01				: BOOL; 
	RGB_Backwards02 			: BOOL; 
	RGB_VertikalDown01			: BOOL; 
	RGB_VertikalDown02			: BOOL; 
	RGB_VertikalUp01			: BOOL;
	RGB_VertikalUp02			: BOOL; 
	RGB_HorizontalForwards01 	: BOOL; 
	RGB_HorizontalForwards02	: BOOL;
	RGB_HorizontalBackwards01 	: BOOL; 
	RGB_HorizontalBackwards02 	: BOOL;
	Init_RGB_Forwards			: BOOL;
	Init_RGB_Backwards			: BOOL;
	Init_RGB_VertikalUp			: BOOL;
	Init_RGB_VertikalDown		: BOOL;
	Init_RGB_HorizontalForwads 	: BOOL;
	Init_RGB_HorizontalBackwards : BOOL;
END_VAR
VAR_OUTPUT
	ConveyorBeltForward: BOOL;
	ConveyorBeltBackward: BOOL;
	RGB_Forwards: BOOL;
	RGB_Backwards: BOOL;
	RGB_VerticalDown: BOOL;
	RGB_VerticalUp: BOOL;
	RGB_HorizontalForward: BOOL;
	RGB_HorizontalBackward: BOOL;
	Light_Q1: BOOL;
	Light_Q2: BOOL;
	Light_Q3: BOOL;
END_VAR
VAR
END_VAR

                   ConveyorBeltForward := ((((((F1) OR (A2))) AND (CB_Forwards))) OR (((Start) AND (F4))));
ConveyorBeltBackward := ((((((F1) OR (A2))) AND (CB_Backwards))) OR (((Start) AND (F4))));
RGB_Forwards := ((((((F1) OR (A2))) AND (((RGB_Forwards01) OR (RGB_Forwards02))))) OR (((Start) AND (F4))) OR (((A6) AND (Init_RGB_Forwards))));
RGB_Backwards := ((((((F1) OR (A2))) AND (((RGB_Backwards01) OR (RGB_Backwards02))))) OR (((Start) AND (F4))) OR (((A6) AND (Init_RGB_Backwards))));
RGB_VerticalDown := ((((((F1) OR (A2))) AND (((RGB_VertikalDown01) OR (RGB_VertikalDown02))))) OR (((Start) AND (F4))) OR (((A6) AND (Init_RGB_VertikalDown))));
RGB_VerticalUp := ((((((F1) OR (A2))) AND (((RGB_VertikalUp01) OR (RGB_VertikalUp02))))) OR (((Start) AND (F4))) OR (((A6) AND (Init_RGB_VertikalUp))));
RGB_HorizontalForward := ((((((F1) OR (A2))) AND (((RGB_HorizontalForwards01) OR (RGB_HorizontalForwards02))))) OR (((Start) AND (F4))) OR (((A6) AND (Init_RGB_HorizontalForwads))));
RGB_HorizontalBackward := ((((((F1) OR (A2))) AND (((RGB_HorizontalBackwards01) OR (RGB_HorizontalBackwards02))))) OR (((Start) AND (F4))) OR (((A6) AND (Init_RGB_HorizontalBackwards))));
Light_Q1 := F1;
Light_Q2 := F4;
Light_Q3 := A1;

                
END_FUNCTION_BLOCK

FUNCTION_BLOCK MBS_ControlOfOutputs
VAR_INPUT
	F4							: BOOL;
	F1							: BOOL;
	A2							: BOOL;
	A1							: BOOL;
	A6							: BOOL;
	Start						: BOOL;
// Output Control
	CB_Forwards 				: BOOL; 
	DmPD_Compressor				: BOOL;
	DmPD_Valve					: BOOL;
	DmPD_RotateCW_VSGtoMR02		: BOOL;	
	DmPD_RotateCW_VSGtoCB		: BOOL;
	DmPD_RotateCW_MR02toCB		: BOOL;
	DmPD_RotateCCW_CBtoMR02		: BOOL;	
	DmPD_RotateCCW_CBtoVSG		: BOOL;
	DmPD_RotateCCW_MR02toVSG	: BOOL;
	MR01_HardeningProcess		: BOOL;
	MR01_HorizontalForwards		: BOOL;
	MR01_HoritzontalBackwards	: BOOL;
	MR01_Compressor				: BOOL;
	MR01_Valve					: BOOL;
	MR02_CuttingProcess			: BOOL;
	VSG_HorizontalForwards		: BOOL;
	VSG_HorizontalBackwards		: BOOL;
	VSG_Valve_VerticalDown		: BOOL;
	VSG_Valve_SuctionToDmPD		: BOOL;
	VSG_Valve_SuctionToMR01		: BOOL;
	VSG_Compressor_VerticalDown : BOOL;
	VSG_Compressor_SuctionToDmPD: BOOL;
	VSG_Compressor_SuctionToMR01: BOOL;
	
// InitDriveMode Output Control	
	Init_DmPD_RotateCCW				: BOOL;
	Init_DmPD_RotateCW				: BOOL;
	Init_MR01_HorizontalForwards	: BOOL;
	Init_MR01_HorizontalBackwards	: BOOL;
	Init_MR02_CuttingProcess		: BOOL;
	Init_VSG_HorizontalForwards		: BOOL;
	Init_VSG_HorizontalBackwards	: BOOL;
END_VAR
VAR_OUTPUT
	ConveyorBeltForward: BOOL;
	CompressorON: BOOL;
	ValveDmPD_ON: BOOL;
	RotateDmPD_CW: BOOL;
	RotateDmPD_CCW: BOOL;
	HardeningProcess : BOOL;
	WorkpieceTableMoveHorizontalForwards : BOOL;
	WorkpieceTableMoveHorizontalBackwards : BOOL;
	ValveMR01_ON : BOOL;
	CuttingProcess_ON : BOOL;
	MoveVSGHorizontalForwards : BOOL;
	MoveVSGHorizontalBackwards : BOOL;
	ValveVSG_VerticalDown_ON : BOOL;
	ValveVSG_Suction_ON : BOOL;
	Light_Q1: BOOL;
	Light_Q2: BOOL;
	Light_Q3: BOOL;
	
END_VAR
VAR
END_VAR

                  ConveyorBeltForward := ((((((F1) OR (A2))) AND (CB_Forwards))) OR (((Start) AND (F4))));
CompressorON := ((((((F1) OR (A2))) AND (((DmPD_Compressor) OR (MR01_Compressor) OR (VSG_Compressor_VerticalDown) OR (VSG_Compressor_SuctionToDmPD) OR (VSG_Compressor_SuctionToMR01))))) OR (((Start) AND (F4))));
ValveDmPD_ON := ((((((F1) OR (A2))) AND (DmPD_Valve))) OR (((Start) AND (F4))));
RotateDmPD_CW := ((((((F1) OR (A2))) AND (((DmPD_RotateCW_VSGtoMR02) OR (DmPD_RotateCW_MR02toCB) OR (DmPD_RotateCW_VSGtoCB))))) OR (((Start) AND (F4))) OR (((A6) AND (Init_DmPD_RotateCW))));
RotateDmPD_CCW := ((((((F1) OR (A2))) AND (((DmPD_RotateCCW_CBtoMR02) OR (DmPD_RotateCCW_CBtoVSG) OR (DmPD_RotateCCW_MR02toVSG))))) OR (((Start) AND (F4))) OR (((A6) AND (Init_DmPD_RotateCCW))));
HardeningProcess := ((((((F1) OR (A2))) AND (MR01_HardeningProcess))) OR (((Start) AND (F4))));
WorkpieceTableMoveHorizontalForwards := ((((((F1) OR (A2))) AND (MR01_HorizontalForwards))) OR (((Start) AND (F4))) OR (((A6) AND (Init_MR01_HorizontalForwards))));
WorkpieceTableMoveHorizontalBackwards := ((((((F1) OR (A2))) AND (MR01_HoritzontalBackwards))) OR (((Start) AND (F4))) OR (((A6) AND (Init_MR01_HorizontalBackwards))));
ValveMR01_ON := ((((((F1) OR (A2))) AND (MR01_Valve))) OR (((Start) AND (F4))));
CuttingProcess_ON := ((((((F1) OR (A2))) AND (MR02_CuttingProcess))) OR (((Start) AND (F4))) OR (((A6) AND (Init_MR02_CuttingProcess))));
MoveVSGHorizontalForwards := ((((((F1) OR (A2))) AND (VSG_HorizontalForwards))) OR (((Start) AND (F4))) OR (((A6) AND (Init_VSG_HorizontalForwards))));
MoveVSGHorizontalBackwards := ((((((F1) OR (A2))) AND (VSG_HorizontalBackwards))) OR (((Start) AND (F4))) OR (((A6) AND (Init_VSG_HorizontalBackwards))));
ValveVSG_VerticalDown_ON := ((((((F1) OR (A2))) AND (VSG_Valve_VerticalDown))) OR (((Start) AND (F4))));
ValveVSG_Suction_ON := ((((((F1) OR (A2))) AND (((VSG_Valve_SuctionToDmPD) OR (VSG_Valve_SuctionToMR01))))) OR (((Start) AND (F4))));
Light_Q1 := F1;
Light_Q2 := F4;
Light_Q3 := A1;

                
END_FUNCTION_BLOCK

FUNCTION_BLOCK SST_ControlOfOutputs
VAR_INPUT
	F4							: BOOL;
	F1							: BOOL;
	A2							: BOOL;
	A1							: BOOL;
	A6							: BOOL;
	Start						: BOOL;	
//Variablen zur Outputsteuerung aus anderen FBs
	//Output-Variablen der Komponente ConveyorBelt	
	CB_MoveForwardToPD01: BOOL;
	CB_MoveForwardToPD02: BOOL;
	CB_MoveForwardToPD03: BOOL;
	CB_MoveForwardTillEnd: BOOL;
	
	//Output-Variablen der Komponente PushingDevice
	PD01_Compressor : BOOL;
	PD02_Compressor : BOOL;
	PD03_Compressor : BOOL;
	PD01_Valve : BOOL;
	PD02_Valve : BOOL;
	PD03_Valve : BOOL;	
	
	//Output-Variablen für Init-Fahrt
	Init_PD01_Compressor : BOOL;
	Init_PD02_Compressor : BOOL;
	Init_PD03_Compressor : BOOL;
	Init_PD01_Valve : BOOL;
	Init_PD02_Valve : BOOL;
	Init_PD03_Valve : BOOL;

END_VAR
VAR_OUTPUT
	ConveyorBeltForward : BOOL;
	CompressorON : BOOL;
	ValvePD01_ON : BOOL;
	ValvePD02_ON : BOOL;
	ValvePD03_ON : BOOL;
	Light_Q1: BOOL;
	Light_Q2: BOOL;
	Light_Q3: BOOL;
	
END_VAR
VAR
END_VAR

                  ConveyorBeltForward := ((((((F1) OR (A2))) AND (((CB_MoveForwardToPD01) OR (CB_MoveForwardToPD02) OR (CB_MoveForwardToPD03) OR (CB_MoveForwardTillEnd))))) OR (((Start) AND (F4))));
CompressorON := ((((((F1) OR (A2))) AND (((PD01_Compressor) OR (PD02_Compressor) OR (PD03_Compressor) OR (Init_PD01_Compressor) OR (Init_PD02_Compressor) OR (Init_PD03_Compressor))))) OR (((Start) AND (F4))));
ValvePD01_ON := ((((((F1) OR (A2))) AND (((PD01_Valve) OR (Init_PD01_Valve))))) OR (((Start) AND (F4))));
ValvePD02_ON := ((((((F1) OR (A2))) AND (((PD02_Valve) OR (Init_PD02_Valve))))) OR (((Start) AND (F4))));
ValvePD03_ON := ((((((F1) OR (A2))) AND (((PD03_Valve) OR (Init_PD03_Valve))))) OR (((Start) AND (F4))));
Light_Q1 := F1;
Light_Q2 := F4;
Light_Q3 := A1;

                
END_FUNCTION_BLOCK

FUNCTION_BLOCK VSG_ControlOfOutputs
VAR_INPUT
	F4							: BOOL;
	F1							: BOOL;
	A2							: BOOL;
	A1							: BOOL;
	A6							: BOOL;
	Start						: BOOL;
	VSG_VertikalDown01			: BOOL; 
	VSG_VertikalDown02			: BOOL; 
	VSG_VertikalUp01			: BOOL;
	VSG_VertikalUp02			: BOOL; 
	VSG_HorizontalForwards01 	: BOOL; 
	VSG_HorizontalForwards02	: BOOL;
	VSG_HorizontalBackwards01 	: BOOL; 
	VSG_HorizontalBackwards02 	: BOOL;
	VSG_RotationCW01		 	: BOOL; 
	VSG_RotationCW02		 	: BOOL;
	VSG_RotationCCW01		 	: BOOL; 
	VSG_RotationCCW02		 	: BOOL;
	VSG_Compressor				: BOOL;
	VSG_Valve					: BOOL;
	Init_VSG_VertikalUp			: BOOL;
	Init_VSG_VertikalDown		: BOOL;	
	Init_VSG_HorizontalForwards : BOOL;
	Init_VSG_HorizontalBackwards: BOOL;
	Init_VSG_RotationCW			: BOOL;
	Init_VSG_RotationCCW		: BOOL;

END_VAR
VAR_OUTPUT
	MoveVerticalDown : BOOL;
	MoveVerticalUp : BOOL;
	MoveHorizontalForwards : BOOL;
	MoveHorizontalBackwards : BOOL;
	MoveRotationCW	: BOOL;
	MoveRotationCCW : BOOL;
	CompressorON : BOOL;
	ValveON : BOOL;
	Light_Q1: BOOL;
	Light_Q2: BOOL;
	Light_Q3: BOOL;
END_VAR
VAR
END_VAR

                  MoveVerticalDown := ((((((F1) OR (A2))) AND (((VSG_VertikalDown01) OR (VSG_VertikalDown02) OR (Init_VSG_VertikalDown))))) OR (((Start) AND (F4))));
MoveVerticalUp := ((((((F1) OR (A2))) AND (((VSG_VertikalUp01) OR (VSG_VertikalUp02) OR (Init_VSG_VertikalUp))))) OR (((Start) AND (F4))));
MoveHorizontalForwards := ((((((F1) OR (A2))) AND (((VSG_HorizontalForwards01) OR (VSG_HorizontalForwards02) OR (Init_VSG_HorizontalForwards))))) OR (((Start) AND (F4))));
MoveHorizontalBackwards := ((((((F1) OR (A2))) AND (((VSG_HorizontalBackwards01) OR (VSG_HorizontalBackwards02) OR (Init_VSG_HorizontalBackwards))))) OR (((Start) AND (F4))));
MoveRotationCW := ((((((F1) OR (A2))) AND (((VSG_RotationCW01) OR (VSG_RotationCW02) OR (Init_VSG_RotationCW))))) OR (((Start) AND (F4))));
MoveRotationCCW := ((((((F1) OR (A2))) AND (((VSG_RotationCCW01) OR (VSG_RotationCCW02) OR (Init_VSG_RotationCCW))))) OR (((Start) AND (F4))));
CompressorON := ((((((F1) OR (A2))) AND (VSG_Compressor))) OR (((Start) AND (F4))));
ValveON := ((((((F1) OR (A2))) AND (VSG_Valve))) OR (((Start) AND (F4))));
Light_Q1 := F1;
Light_Q2 := F4;
Light_Q3 := A1;

                
END_FUNCTION_BLOCK

FUNCTION_BLOCK HRL_DiagnosisHandler
VAR_INPUT
    Diagnose_gefordert : BOOL;
    ErrorDetectedRaw   : BOOL;
    Reset              : BOOL;
    PulseTime          : TIME := T#100MS;
END_VAR
VAR_OUTPUT
    Err_detected  : BOOL := FALSE;
    Diag_finished : BOOL := FALSE;
    Alt_found     : BOOL := FALSE;
    Busy          : BOOL := FALSE;
END_VAR
VAR
    rtReq      : R_TRIG;
    rtError    : R_TRIG;
    rtDiagAck  : R_TRIG;
    rtAltFound : R_TRIG;
    tpPulse    : TP;
END_VAR

                  rtReq(CLK := Diagnose_gefordert);
rtError(CLK := ErrorDetectedRaw);
rtDiagAck(CLK := OPCUA.Diag_finished);
rtAltFound(CLK := OPCUA.Alt_found);

IF Reset THEN
    Err_detected := FALSE;
    Diag_finished := FALSE;
    Alt_found := FALSE;
    Busy := FALSE;
    OPCUA.TriggerD2 := FALSE;
END_IF

IF rtError.Q THEN
    Err_detected := TRUE;
    Diag_finished := FALSE;
    Alt_found := FALSE;
END_IF

tpPulse(
    IN := rtReq.Q AND Err_detected AND NOT Busy,
    PT := PulseTime
);

IF rtReq.Q AND Err_detected AND NOT Busy THEN
    Busy := TRUE;
END_IF

IF tpPulse.Q THEN
    OPCUA.TriggerD2 := TRUE;
ELSIF OPCUA.TriggerD2 AND Diag_finished THEN
    OPCUA.TriggerD2 := FALSE;
END_IF

IF Busy AND rtDiagAck.Q THEN
    Diag_finished := TRUE;
    Alt_found := FALSE;
    Busy := FALSE;
    OPCUA.Diag_finished := FALSE;
    OPCUA.TriggerD2 := FALSE;
END_IF

IF Busy AND rtAltFound.Q THEN
    Alt_found := TRUE;
    Diag_finished := TRUE;
    Busy := FALSE;
    OPCUA.Alt_found := FALSE;
    OPCUA.TriggerD2 := FALSE;
END_IF

IF NOT Diagnose_gefordert AND (Diag_finished OR Alt_found) THEN
    Err_detected := FALSE;
    Diag_finished := FALSE;
    Alt_found := FALSE;
END_IF

                
END_FUNCTION_BLOCK

FUNCTION_BLOCK VSG_DiagnosisHandler
VAR_INPUT
    Diagnose_gefordert : BOOL;
    ErrorDetectedRaw   : BOOL;
    Reset              : BOOL;
    PulseTime          : TIME := T#100MS;
END_VAR
VAR_OUTPUT
    Err_detected  : BOOL := FALSE;
    Diag_finished : BOOL := FALSE;
    Alt_found     : BOOL := FALSE;
    Busy          : BOOL := FALSE;
END_VAR
VAR
    rtReq      : R_TRIG;
    rtError    : R_TRIG;
    rtDiagAck  : R_TRIG;
    rtAltFound : R_TRIG;
    tpPulse    : TP;
END_VAR

                  rtReq(CLK := Diagnose_gefordert);
rtError(CLK := ErrorDetectedRaw);
rtDiagAck(CLK := OPCUA.Diag_finished);
rtAltFound(CLK := OPCUA.Alt_found);

IF Reset THEN
    Err_detected := FALSE;
    Diag_finished := FALSE;
    Alt_found := FALSE;
    Busy := FALSE;
    OPCUA.TriggerD2 := FALSE;
END_IF

IF rtError.Q THEN
    Err_detected := TRUE;
    Diag_finished := FALSE;
    Alt_found := FALSE;
	OPCUA.TriggerD2 := TRUE;
END_IF

IF rtReq.Q AND Err_detected AND NOT Busy THEN
    Busy := TRUE;
END_IF

IF OPCUA.TriggerD2 AND Diag_finished THEN
    OPCUA.TriggerD2 := FALSE;
END_IF

IF Busy AND rtDiagAck.Q THEN
    Diag_finished := TRUE;
    Alt_found := FALSE;
    Busy := FALSE;
    OPCUA.Diag_finished := FALSE;
    OPCUA.TriggerD2 := FALSE;
END_IF

IF Busy AND rtAltFound.Q THEN
    Alt_found := TRUE;
    Diag_finished := TRUE;
    Busy := FALSE;
    OPCUA.Alt_found := FALSE;
    OPCUA.TriggerD2 := FALSE;
END_IF

IF NOT Diagnose_gefordert AND (Diag_finished OR Alt_found) THEN
    Err_detected := FALSE;
    Diag_finished := FALSE;
    Alt_found := FALSE;
END_IF

                
END_FUNCTION_BLOCK

FUNCTION_BLOCK HRL_RGB_InitialStateDrive
VAR_INPUT
	MethodCall_InitDrive		: BOOL;
	ESS							: BOOL;
	InputInitDriveMode			: BOOL;
	TouchSensor01_SRM			: BOOL;
	TouchSensor02_RGB_vertical	: BOOL;
	TouchSensor03_RGB_horizontal: BOOL;
	TOF_Time_TSR				: TIME;
	InitDriveMode 				: BOOL;
END_VAR

VAR_OUTPUT
	SRM_MotorBackwards: BOOL;
	SRM_MotorForwards: BOOL;
	RGB_VerticalUp: BOOL;
	RGB_VerticalDown: BOOL;
	RGB_HorizontalForwards: BOOL;
	RGB_HorizontalBackwards: BOOL;
	ResetMethodCall_SRM	: BOOL;
	ResetMethodCall_RGB_Vertical	: BOOL;
	ResetMethodCall_RGB_Horizontal	: BOOL;
	Count_SRM_MotorBackw : INT;
	Count_SRM_MotorForw : INT;
END_VAR
VAR
	TSR : BOOL := TRUE;
	DirectionVerticalSRM : BOOL := TRUE;
	DirectionVertical : BOOL := TRUE;
	DirectionHorizontal : BOOL := TRUE;
	
	HRL_RGB_SRM_InitDrive: AxisControl_MultipleInputSensors;
	HRL_RGB_Vertical_InitDrive: AxisControl_MultipleInputSensors;
	HRL_RGB_Horizontal_InitDrive: AxisControl_MultipleInputSensors;
END_VAR

                  HRL_RGB_SRM_InitDrive(
    MethodCall := MethodCall_InitDrive,
    EmergencyStopSignal := ESS,
    Direction := DirectionVerticalSRM,
    InitStateDrive_Input := InputInitDriveMode,
    DI01 := FALSE,
    DI02 := TouchSensor01_SRM,
    TouchSensorRelief := TSR,
    TOF_Time_MotorControl := T#0MS,
    TOF_Time_TouchSensorRelief := TOF_Time_TSR,
    OperatingMode := InitDriveMode
);
SRM_MotorBackwards := HRL_RGB_SRM_InitDrive.DigitalOutputControl_01;

HRL_RGB_Vertical_InitDrive(
    MethodCall := MethodCall_InitDrive,
    EmergencyStopSignal := ESS,
    Direction := DirectionVertical,
    InitStateDrive_Input := InputInitDriveMode,
    DI01 := FALSE,
    DI02 := TouchSensor02_RGB_vertical,
    TouchSensorRelief := TSR,
    TOF_Time_MotorControl := T#0MS,
    TOF_Time_TouchSensorRelief := TOF_Time_TSR,
    OperatingMode := InitDriveMode
);
RGB_VerticalUp := HRL_RGB_Vertical_InitDrive.DigitalOutputControl_01;

HRL_RGB_Horizontal_InitDrive(
    MethodCall := MethodCall_InitDrive,
    EmergencyStopSignal := ESS,
    Direction := DirectionHorizontal,
    InitStateDrive_Input := InputInitDriveMode,
    DI01 := FALSE,
    DI02 := TouchSensor03_RGB_horizontal,
    TouchSensorRelief := TSR,
    TOF_Time_MotorControl := T#0MS,
    TOF_Time_TouchSensorRelief := TOF_Time_TSR,
    OperatingMode := InitDriveMode
);
RGB_HorizontalBackwards := HRL_RGB_Horizontal_InitDrive.DigitalOutputControl_01;
                
END_FUNCTION_BLOCK

FUNCTION_BLOCK MBS_DmPD_InitialStateDrive
VAR_INPUT
	MethodCall_InitDrive : BOOL;
	ESS : BOOL;
	InputInitialStateDrive : BOOL;
	DI02_CW : BOOL;
	DI01_CCW : BOOL;
	DI02_CCW : BOOL;	
	InitDriveMode : BOOL;
END_VAR
VAR_OUTPUT
	MotorControl_CW : BOOL;
	MotorControl_CCW : BOOL;
	ResetMethodCallRotateCW : BOOL;
	ResetMethodCallRotateCCW : BOOL;
END_VAR
VAR
	DirectionCW : STRING;
	DirectionCCW : STRING;
	MBS_DmPD_InitDrive_Rotate_CW: AxisControl_MultipleInputSensors;
	MBS_DmPD_InitDrive_Rotate_CCW: AxisControl_MultipleInputSensors;
END_VAR

                  MBS_DmPD_InitDrive_Rotate_CW(
    MethodCall := MethodCall_InitDrive,
    EmergencyStopSignal := ESS,
    Direction := DirectionCW,
    InitStateDrive_Input := InputInitialStateDrive,
    DI01 := ,
    DI02 := DI02_CW,
    TouchSensorRelief := ,
    TOF_Time_MotorControl := ,
    TOF_Time_TouchSensorRelief := ,
    OperatingMode := InitDriveMode
);
MotorControl_CW := MBS_DmPD_InitDrive_Rotate_CW.DigitalOutputControl_01;
MBS_DmPD_InitDrive_Rotate_CCW(
    MethodCall := MethodCall_InitDrive,
    EmergencyStopSignal := ESS,
    Direction := DirectionCCW,
    InitStateDrive_Input := ,
    DI01 := DI01_CCW,
    DI02 := DI02_CCW,
    TouchSensorRelief := ,
    TOF_Time_MotorControl := ,
    TOF_Time_TouchSensorRelief := ,
    OperatingMode := InitDriveMode
);
MotorControl_CCW := MBS_DmPD_InitDrive_Rotate_CCW.DigitalOutputControl_01;

                
END_FUNCTION_BLOCK

FUNCTION_BLOCK MBS_MR01_InitialStateDrive
VAR_INPUT
	MethodCall_InitDrive : BOOL;
	ESS : BOOL;
	InputInitStateDrive : BOOL;
	TouchSensor01 : BOOL;
	TouchSensor02 : BOOL;
	InitDriveMode : BOOL;
END_VAR
VAR_OUTPUT
	MotorControlHorizontalForwards : BOOL;
	MotorControlHorizontalBackwards : BOOL;
	ResetMethodCallInitDriveMR01_Backwards : BOOL;
	ResetMethodCallInitDriveMR01_Forwards : BOOL;
END_VAR
VAR
	DirectionHorizontal : STRING;
	
	MBS_MR01_InitDrive_HorizontalForwards: AxisControl_MultipleInputSensors;
	MBS_MR01_InitDrive_HorizontalBackwards: AxisControl_MultipleInputSensors;
END_VAR

                  MBS_MR01_InitDrive_HorizontalBackwards(
    MethodCall := MethodCall_InitDrive,
    EmergencyStopSignal := ESS,
    Direction := DirectionHorizontal,
    InitStateDrive_Input := InputInitStateDrive,
    DI01 := ,
    DI02 := TouchSensor01,
    TouchSensorRelief := ,
    TOF_Time_MotorControl := ,
    TOF_Time_TouchSensorRelief := ,
    OperatingMode := InitDriveMode
);
MotorControlHorizontalBackwards := MBS_MR01_InitDrive_HorizontalBackwards.DigitalOutputControl_01;
MBS_MR01_InitDrive_HorizontalForwards(
    MethodCall := MethodCall_InitDrive,
    EmergencyStopSignal := ESS,
    Direction := DirectionHorizontal,
    InitStateDrive_Input := ,
    DI01 := TouchSensor01,
    DI02 := TouchSensor02,
    TouchSensorRelief := ,
    TOF_Time_MotorControl := ,
    TOF_Time_TouchSensorRelief := ,
    OperatingMode := InitDriveMode
);
MotorControlHorizontalForwards := MBS_MR01_InitDrive_HorizontalForwards.DigitalOutputControl_01;

                
END_FUNCTION_BLOCK

FUNCTION_BLOCK MBS_MR02_InitialStateDrive
VAR_INPUT
	MethodCall_InitDrive : BOOL;
	ESS : BOOL;
	InputInitialStateDrive : BOOL;
	TOF_Time_InitCuttingTime : TIME;
	InitDriveMode : BOOL;
END_VAR
VAR_OUTPUT
	CheckMR02MotorControl : BOOL;
	ResetMethodCallCuttingProcess : BOOL;
END_VAR
VAR
	MBS_MR02_InitDrive_CuttingProcess: CuttingProcess;
END_VAR

                  MBS_MR02_InitDrive_CuttingProcess(
    MethodCall := MethodCall_InitDrive,
    EmergencyStopSignal := ESS,
    InitStateDrive_Input := InputInitialStateDrive,
    DI01 := ,
    TOF_Time_CuttingTime := TOF_Time_InitCuttingTime,
    OperatingMode := InitDriveMode
);
CheckMR02MotorControl := MBS_MR02_InitDrive_CuttingProcess.DigitalOutputControl_01;

                
END_FUNCTION_BLOCK

FUNCTION_BLOCK MBS_VSG_InitialStateDrive
VAR_INPUT
	MethodCall_InitDrive : BOOL;
	ESS : BOOL;
	InputInitStateDrive : BOOL;
	TouchSensor01 : BOOL;
	TOF_Time_TSR : TIME;
	InitDriveMode : BOOL;	
END_VAR

VAR_OUTPUT
	DO_HorizontalMoveInitDriveVSG_01 : BOOL;
	DO_HorizontalMoveInitDriveVSG_02 : BOOL;
	ResetMethodCallInitDriveVSG : BOOL;
END_VAR

VAR
	TSR : BOOL := TRUE;
	DirectionHorizontal : STRING;

	MBS_VSG_InitDrive: AxisControl_MultipleInputSensors;
END_VAR

                  MBS_VSG_InitDrive(
    MethodCall := MethodCall_InitDrive,
    EmergencyStopSignal := ESS,
    Direction := DirectionHorizontal,
    InitStateDrive_Input := InputInitStateDrive,
    DI01 := ,
    DI02 := TouchSensor01,
    TouchSensorRelief := TSR,
    TOF_Time_MotorControl := ,
    TOF_Time_TouchSensorRelief := TOF_Time_TSR,
    OperatingMode := InitDriveMode
);
DO_HorizontalMoveInitDriveVSG_01 := MBS_VSG_InitDrive.DigitalOutputControl_01;

                
END_FUNCTION_BLOCK

FUNCTION_BLOCK SST_PD_InitialStateDrive
VAR_INPUT
	MethodCall_InitDrive : BOOL;
	ESS : BOOL;
	InputInitialStateDrive : BOOL;
	TON_Time_PowerOFFSelfSet : TIME;
	InitDriveMode : BOOL;
END_VAR
VAR_OUTPUT
	MotorControl_PD01_Compressor : BOOL;
	MotorControl_PD01_Valve : BOOL;
	MotorControl_PD02_Compressor : BOOL;
	MotorControl_PD02_Valve : BOOL;
	MotorControl_PD03_Compressor : BOOL;
	MotorControl_PD03_Valve : BOOL;
	ResetMethodCallMovePD01 : BOOL;
	ResetMethodCallMovePD02 : BOOL;
	ResetMethodCallMovePD03 : BOOL;
END_VAR
VAR
	DestinationHorizontal : STRING;
	PowerOfF_SelfSet : BOOL := TRUE;
	SST_PD01_InitDrive : CompressorControl;
	SST_PD02_InitDrive : CompressorControl;
	SST_PD03_InitDrive : CompressorControl;
END_VAR

                  SST_PD01_InitDrive(
    MethodCall := MethodCall_InitDrive,
    EmergencyStopSignal := ESS,
    Destination := DestinationHorizontal,
    InitStateDrive_Input := InputInitialStateDrive,
    DI01 := ,
    DI02 := ,
    DI03_EncoderStart01 := ,
    DI04_EncoderStart02 := ,
    DI05_EncoderStart03 := ,
    DI06_EncoderStart04 := ,
    DI07_EncoderStart05 := ,
    DI08_EncoderStart06 := ,
    DI09_EncoderTarget01 := ,
    DI10_EncoderTarget02 := ,
    DI11_EncoderTarget03 := ,
    DI12_EncoderTarget04 := ,
    DI13_EncoderTarget05 := ,
    DI14_EncoderTarget06 := ,
    PowerOFF_SelfSet := PowerOfF_SelfSet,
    TON_Time_PowerOFFSelfSet := TON_Time_PowerOFFSelfSet,
    TON_Time_Compressor := PowerOnDelay_Compressor,
    TON_Time_Valve := PowerOnDelay_Valve,
    OperatingMode := AutomaticMode
);
MotorControl_PD01_Compressor := SST_PD01_InitDrive.DigitalOutputControl_01;
SST_PD02_InitDrive(
    MethodCall := MethodCall_InitDrive,
    EmergencyStopSignal := ESS,
    Destination := DestinationHorizontal,
    InitStateDrive_Input := InputInitialStateDrive,
    DI01 := ,
    DI02 := ,
    DI03_EncoderStart01 := ,
    DI04_EncoderStart02 := ,
    DI05_EncoderStart03 := ,
    DI06_EncoderStart04 := ,
    DI07_EncoderStart05 := ,
    DI08_EncoderStart06 := ,
    DI09_EncoderTarget01 := ,
    DI10_EncoderTarget02 := ,
    DI11_EncoderTarget03 := ,
    DI12_EncoderTarget04 := ,
    DI13_EncoderTarget05 := ,
    DI14_EncoderTarget06 := ,
    PowerOFF_SelfSet := PowerOfF_SelfSet,
    TON_Time_PowerOFFSelfSet := TON_Time_PowerOFFSelfSet,
    TON_Time_Compressor := PowerOnDelay_Compressor,
    TON_Time_Valve := PowerOnDelay_Valve,
    OperatingMode := AutomaticMode
);
MotorControl_PD02_Compressor := SST_PD02_InitDrive.DigitalOutputControl_01;
SST_PD03_InitDrive(
    MethodCall := MethodCall_InitDrive,
    EmergencyStopSignal := ESS,
    Destination := DestinationHorizontal,
    InitStateDrive_Input := InputInitialStateDrive,
    DI01 := ,
    DI02 := ,
    DI03_EncoderStart01 := ,
    DI04_EncoderStart02 := ,
    DI05_EncoderStart03 := ,
    DI06_EncoderStart04 := ,
    DI07_EncoderStart05 := ,
    DI08_EncoderStart06 := ,
    DI09_EncoderTarget01 := ,
    DI10_EncoderTarget02 := ,
    DI11_EncoderTarget03 := ,
    DI12_EncoderTarget04 := ,
    DI13_EncoderTarget05 := ,
    DI14_EncoderTarget06 := ,
    PowerOFF_SelfSet := PowerOfF_SelfSet,
    TON_Time_PowerOFFSelfSet := TON_Time_PowerOFFSelfSet,
    TON_Time_Compressor := PowerOnDelay_Compressor,
    TON_Time_Valve := PowerOnDelay_Valve,
    OperatingMode := AutomaticMode
);
MotorControl_PD03_Compressor := SST_PD03_InitDrive.DigitalOutputControl_01;
                
END_FUNCTION_BLOCK

FUNCTION_BLOCK VSG_InitialStateDrive
VAR_INPUT
    MethodCall_InitDrive : BOOL;
    ESS : BOOL;
    InputInitDriveMode : BOOL;

    TouchSensor01_Rotation : BOOL;
    TouchSensor02_Vertical : BOOL;
    TouchSensor03_horizontal : BOOL;

    TOF_Time_TSR : TIME;
    InitDriveMode : BOOL;
END_VAR

VAR_OUTPUT
    VSG_Init_RotateCW : BOOL;
    VSG_Init_RotateCCW : BOOL;

    VSG_Init_VerticalUp : BOOL;
    VSG_Init_VerticalDown : BOOL;

    VSG_Init_HorizontalForwards : BOOL;
    VSG_Init_HorizontalBackwards : BOOL;

    ResetMethodCall_RotateCW : BOOL;
    ResetMethodCall_RGB_Vertical : BOOL;
    ResetMethodCall_RGB_Horizontal : BOOL;
END_VAR

VAR
    TSR : BOOL := TRUE;

    DirectionVertical : BOOL := TRUE;
    DirectionHorizontal : BOOL := TRUE;
    DirectionRotation : BOOL := TRUE;

    VSG_InitDrive_Rotate_CW : AxisControl_MultipleInputSensors;
    VSG_InitDrive_Vertical_Up : AxisControl_MultipleInputSensors;
    VSG_InitDrive_Horizontal_Backwards : AxisControl_MultipleInputSensors;
END_VAR

                  VSG_InitDrive_Rotate_CW(
    MethodCall := MethodCall_InitDrive,
    EmergencyStopSignal := NOT ESS,
    Direction := DirectionRotation,
    InitStateDrive_Input := InputInitDriveMode,
    DI01 := FALSE,
    DI02 := TouchSensor01_Rotation,
    TouchSensorRelief := TSR,
    TOF_Time_MotorControl := T#0MS,
    TOF_Time_TouchSensorRelief := TOF_Time_TSR,
    OperatingMode := InitDriveMode
);

VSG_Init_RotateCW := VSG_InitDrive_Rotate_CW.DigitalOutputControl_01;
VSG_Init_RotateCCW := FALSE;
ResetMethodCall_RotateCW := VSG_InitDrive_Rotate_CW.ResetMethodCall;


VSG_InitDrive_Vertical_Up(
    MethodCall := MethodCall_InitDrive,
    EmergencyStopSignal := NOT ESS,
    Direction := DirectionVertical,
    InitStateDrive_Input := InputInitDriveMode,
    DI01 := FALSE,
    DI02 := TouchSensor02_Vertical,
    TouchSensorRelief := TSR,
    TOF_Time_MotorControl := T#0MS,
    TOF_Time_TouchSensorRelief := TOF_Time_TSR,
    OperatingMode := InitDriveMode
);

VSG_Init_VerticalUp := VSG_InitDrive_Vertical_Up.DigitalOutputControl_01;
VSG_Init_VerticalDown := FALSE;
ResetMethodCall_RGB_Vertical := VSG_InitDrive_Vertical_Up.ResetMethodCall;


VSG_InitDrive_Horizontal_Backwards(
    MethodCall := MethodCall_InitDrive,
    EmergencyStopSignal := NOT ESS,
    Direction := DirectionHorizontal,
    InitStateDrive_Input := InputInitDriveMode,
    DI01 := FALSE,
    DI02 := TouchSensor03_horizontal,
    TouchSensorRelief := TSR,
    TOF_Time_MotorControl := T#0MS,
    TOF_Time_TouchSensorRelief := TOF_Time_TSR,
    OperatingMode := InitDriveMode
);

VSG_Init_HorizontalForwards := FALSE;
VSG_Init_HorizontalBackwards := VSG_InitDrive_Horizontal_Backwards.DigitalOutputControl_01;
ResetMethodCall_RGB_Horizontal := VSG_InitDrive_Horizontal_Backwards.ResetMethodCall;
                
END_FUNCTION_BLOCK

FUNCTION_BLOCK PUBLIC FB_MyOpcUaMethod
VAR_INPUT
	in1 : INT;
	in2 : INT;
END_VAR
VAR_OUTPUT
	result : INT;
END_VAR

                  
                

{attribute 'TcRpcEnable' := '1'}
METHOD PUBLIC Multiply : INT
VAR_INPUT
	a : INT;
	b : INT;
END_VAR
                        Multiply := a * b;
                      
END_METHOD
END_FUNCTION_BLOCK

{attribute 'OPC.UA.DA.JobMethod' := 'JobMethode_Schablone'}
FUNCTION_BLOCK JobMethode_Schablone
VAR
	AlwaysTrue : BOOL := TRUE;
	// Used for debugging purposes to display InputArguments of method call
	MethodCall_Name : BOOL := FALSE; // used to store InputArg "MethodCall" from Start() method
	Direction_01 : BOOL := FALSE;
	Direction_02 : BOOL := FALSE;
	TS_EndschalterEntlastung : BOOL;
	callCounterStart : ULINT; // counts how many times the Start() method has been called
	callCounterCheckState : ULINT; // counts how many times the CheckState() method has been called
	callCounterAbort : ULINT; // counts how many times the Abort() method has been called
	
	// Variables to determine if a job has been started (Start() method has been called) or finished
	jobRunning : BOOL;
	jobFinished : BOOL;

	// State machine variable
	state : UDINT;
	
	//Variablen des Transport FBs
	ResetCall : BOOL := FALSE;	
	JobMethode_Name : AxisControl_MultipleInputSensors;
END_VAR
	
VAR_INPUT
	NotAusSignal: BOOL;
	LightSensor_01 : BOOL;
	LightSensor_02 : BOOL;
	TS_Endschalter_01 : BOOL;
	TS_Endschalter_02 : BOOL;
	TOF_Time_Motoransteuerung : TIME;
	TOF_Time_EndschalterEntlastung : TIME;
END_VAR

VAR_OUTPUT
	Motor_Ansteuerung01 : BOOL;
	Motor_Ansteuerung02 : BOOL;
END_VAR

                  JobMethode_Name(
    MethodCall := MethodCall_Name,
    NotAus_Signal := NotAusSignal,
    Direction_01 := Direction_01,
    Direction_02 := Direction_02,
    LightSensor_01 := LightSensor_01,
    LightSensor_02 := LightSensor_02,
    TS_Endschalter_01 := TS_Endschalter_01,
    AutomaticMode := _REFACTOR_,
    TS_Endschalter_02 := TS_Endschalter_02,
    TS_EndschalterEntlastung := TS_EndschalterEntlastung,
    TOF_Time_Motoransteuerung := TOF_Time_Motoransteuerung,
    TOF_Time_EndschalterEntlastung := TOF_Time_EndschalterEntlastung
);
Motor_Ansteuerung01 := JobMethode_Name.Motor_Direction01;

                

{attribute 'TcRpcEnable' := '1'}
METHOD Abort : HRESULT
VAR_INPUT
	hdl : UDINT; // Do not change, used by server.
END_VAR
                        callCounterAbort := callCounterAbort + 1;
                      
END_METHOD

